	bArm1VertStn4AglDown_00 AT %MX25416.0 : BOOL;
	bArm1VertStn4AglDown_01 AT %MX25416.1 : BOOL;
	bArm1VertStn4AglDown_02 AT %MX25416.2 : BOOL;
	bArm1VertStn4AglDown_03 AT %MX25416.3 : BOOL;
	bArm1VertStn4AglDown_04 AT %MX25416.4 : BOOL;
	bArm1VertStn4AglDown_05 AT %MX25416.5 : BOOL;
	bArm1VertStn4AglDown_06 AT %MX25416.6 : BOOL;
	bArm1VertStn4AglDown_07 AT %MX25416.7 : BOOL;
	bArm1VertStn4AglDown_08 AT %MX25416.8 : BOOL;
	bArm1VertStn4AglDown_09 AT %MX25416.9 : BOOL;
	bArm1VertStn4AglDown_10 AT %MX25416.10 : BOOL;
	bArm1VertStn4AglDown_11 AT %MX25416.11 : BOOL;
	bArm1VertStn4AglDown_12 AT %MX25416.12 : BOOL;
	bArm1VertStn4AglDown_13 AT %MX25416.13 : BOOL;
	bArm1VertStn4AglDown_14 AT %MX25416.14 : BOOL;
	bArm1VertStn4AglDown_15 AT %MX25416.15 : BOOL;
	bArm1VertStn4AglDown_16 AT %MX25416.16 : BOOL;
	bArm1VertStn4AglDown_17 AT %MX25416.17 : BOOL;
	bArm1VertStn4AglDown_18 AT %MX25416.18 : BOOL;
	bArm1VertStn4AglDown_19 AT %MX25416.19 : BOOL;
	bArm1VertStn4AglDown_20 AT %MX25416.20 : BOOL;
	bArm1VertStn4AglDown_21 AT %MX25416.21 : BOOL;
	bArm1VertStn4AglDown_22 AT %MX25416.22 : BOOL;
	bArm1VertStn4AglDown_23 AT %MX25416.23 : BOOL;
	bArm1VertStn4AglDown_24 AT %MX25416.24 : BOOL;
	bArm1VertStn4AglDown_25 AT %MX25416.25 : BOOL;
	bArm1VertStn4AglDown_26 AT %MX25416.26 : BOOL;
	bArm1VertStn4AglDown_27 AT %MX25416.27 : BOOL;
	bArm1VertStn4AglDown_28 AT %MX25416.28 : BOOL;
	bArm1VertStn4AglDown_29 AT %MX25416.29 : BOOL;
	bArm1VertStn4AglDown_30 AT %MX25416.30 : BOOL;
	bArm1VertStn4AglDown_31 AT %MX25416.31 : BOOL;

	bArm1VertStn5AglDown_00 AT %MX25420.0 : BOOL;
	bArm1VertStn5AglDown_01 AT %MX25420.1 : BOOL;
	bArm1VertStn5AglDown_02 AT %MX25420.2 : BOOL;
	bArm1VertStn5AglDown_03 AT %MX25420.3 : BOOL;
	bArm1VertStn5AglDown_04 AT %MX25420.4 : BOOL;
	bArm1VertStn5AglDown_05 AT %MX25420.5 : BOOL;
	bArm1VertStn5AglDown_06 AT %MX25420.6 : BOOL;
	bArm1VertStn5AglDown_07 AT %MX25420.7 : BOOL;
	bArm1VertStn5AglDown_08 AT %MX25420.8 : BOOL;
	bArm1VertStn5AglDown_09 AT %MX25420.9 : BOOL;
	bArm1VertStn5AglDown_10 AT %MX25420.10 : BOOL;
	bArm1VertStn5AglDown_11 AT %MX25420.11 : BOOL;
	bArm1VertStn5AglDown_12 AT %MX25420.12 : BOOL;
	bArm1VertStn5AglDown_13 AT %MX25420.13 : BOOL;
	bArm1VertStn5AglDown_14 AT %MX25420.14 : BOOL;
	bArm1VertStn5AglDown_15 AT %MX25420.15 : BOOL;
	bArm1VertStn5AglDown_16 AT %MX25420.16 : BOOL;
	bArm1VertStn5AglDown_17 AT %MX25420.17 : BOOL;
	bArm1VertStn5AglDown_18 AT %MX25420.18 : BOOL;
	bArm1VertStn5AglDown_19 AT %MX25420.19 : BOOL;
	bArm1VertStn5AglDown_20 AT %MX25420.20 : BOOL;
	bArm1VertStn5AglDown_21 AT %MX25420.21 : BOOL;
	bArm1VertStn5AglDown_22 AT %MX25420.22 : BOOL;
	bArm1VertStn5AglDown_23 AT %MX25420.23 : BOOL;
	bArm1VertStn5AglDown_24 AT %MX25420.24 : BOOL;
	bArm1VertStn5AglDown_25 AT %MX25420.25 : BOOL;
	bArm1VertStn5AglDown_26 AT %MX25420.26 : BOOL;
	bArm1VertStn5AglDown_27 AT %MX25420.27 : BOOL;
	bArm1VertStn5AglDown_28 AT %MX25420.28 : BOOL;
	bArm1VertStn5AglDown_29 AT %MX25420.29 : BOOL;
	bArm1VertStn5AglDown_30 AT %MX25420.30 : BOOL;
	bArm1VertStn5AglDown_31 AT %MX25420.31 : BOOL;

	bArm1VertStn6AglDown_00 AT %MX25424.0 : BOOL;
	bArm1VertStn6AglDown_01 AT %MX25424.1 : BOOL;
	bArm1VertStn6AglDown_02 AT %MX25424.2 : BOOL;
	bArm1VertStn6AglDown_03 AT %MX25424.3 : BOOL;
	bArm1VertStn6AglDown_04 AT %MX25424.4 : BOOL;
	bArm1VertStn6AglDown_05 AT %MX25424.5 : BOOL;
	bArm1VertStn6AglDown_06 AT %MX25424.6 : BOOL;
	bArm1VertStn6AglDown_07 AT %MX25424.7 : BOOL;
	bArm1VertStn6AglDown_08 AT %MX25424.8 : BOOL;
	bArm1VertStn6AglDown_09 AT %MX25424.9 : BOOL;
	bArm1VertStn6AglDown_10 AT %MX25424.10 : BOOL;
	bArm1VertStn6AglDown_11 AT %MX25424.11 : BOOL;
	bArm1VertStn6AglDown_12 AT %MX25424.12 : BOOL;
	bArm1VertStn6AglDown_13 AT %MX25424.13 : BOOL;
	bArm1VertStn6AglDown_14 AT %MX25424.14 : BOOL;
	bArm1VertStn6AglDown_15 AT %MX25424.15 : BOOL;
	bArm1VertStn6AglDown_16 AT %MX25424.16 : BOOL;
	bArm1VertStn6AglDown_17 AT %MX25424.17 : BOOL;
	bArm1VertStn6AglDown_18 AT %MX25424.18 : BOOL;
	bArm1VertStn6AglDown_19 AT %MX25424.19 : BOOL;
	bArm1VertStn6AglDown_20 AT %MX25424.20 : BOOL;
	bArm1VertStn6AglDown_21 AT %MX25424.21 : BOOL;
	bArm1VertStn6AglDown_22 AT %MX25424.22 : BOOL;
	bArm1VertStn6AglDown_23 AT %MX25424.23 : BOOL;
	bArm1VertStn6AglDown_24 AT %MX25424.24 : BOOL;
	bArm1VertStn6AglDown_25 AT %MX25424.25 : BOOL;
	bArm1VertStn6AglDown_26 AT %MX25424.26 : BOOL;
	bArm1VertStn6AglDown_27 AT %MX25424.27 : BOOL;
	bArm1VertStn6AglDown_28 AT %MX25424.28 : BOOL;
	bArm1VertStn6AglDown_29 AT %MX25424.29 : BOOL;
	bArm1VertStn6AglDown_30 AT %MX25424.30 : BOOL;
	bArm1VertStn6AglDown_31 AT %MX25424.31 : BOOL;

	bArm1VertStn7AglDown_00 AT %MX25428.0 : BOOL;
	bArm1VertStn7AglDown_01 AT %MX25428.1 : BOOL;
	bArm1VertStn7AglDown_02 AT %MX25428.2 : BOOL;
	bArm1VertStn7AglDown_03 AT %MX25428.3 : BOOL;
	bArm1VertStn7AglDown_04 AT %MX25428.4 : BOOL;
	bArm1VertStn7AglDown_05 AT %MX25428.5 : BOOL;
	bArm1VertStn7AglDown_06 AT %MX25428.6 : BOOL;
	bArm1VertStn7AglDown_07 AT %MX25428.7 : BOOL;
	bArm1VertStn7AglDown_08 AT %MX25428.8 : BOOL;
	bArm1VertStn7AglDown_09 AT %MX25428.9 : BOOL;
	bArm1VertStn7AglDown_10 AT %MX25428.10 : BOOL;
	bArm1VertStn7AglDown_11 AT %MX25428.11 : BOOL;
	bArm1VertStn7AglDown_12 AT %MX25428.12 : BOOL;
	bArm1VertStn7AglDown_13 AT %MX25428.13 : BOOL;
	bArm1VertStn7AglDown_14 AT %MX25428.14 : BOOL;
	bArm1VertStn7AglDown_15 AT %MX25428.15 : BOOL;
	bArm1VertStn7AglDown_16 AT %MX25428.16 : BOOL;
	bArm1VertStn7AglDown_17 AT %MX25428.17 : BOOL;
	bArm1VertStn7AglDown_18 AT %MX25428.18 : BOOL;
	bArm1VertStn7AglDown_19 AT %MX25428.19 : BOOL;
	bArm1VertStn7AglDown_20 AT %MX25428.20 : BOOL;
	bArm1VertStn7AglDown_21 AT %MX25428.21 : BOOL;
	bArm1VertStn7AglDown_22 AT %MX25428.22 : BOOL;
	bArm1VertStn7AglDown_23 AT %MX25428.23 : BOOL;
	bArm1VertStn7AglDown_24 AT %MX25428.24 : BOOL;
	bArm1VertStn7AglDown_25 AT %MX25428.25 : BOOL;
	bArm1VertStn7AglDown_26 AT %MX25428.26 : BOOL;
	bArm1VertStn7AglDown_27 AT %MX25428.27 : BOOL;
	bArm1VertStn7AglDown_28 AT %MX25428.28 : BOOL;
	bArm1VertStn7AglDown_29 AT %MX25428.29 : BOOL;
	bArm1VertStn7AglDown_30 AT %MX25428.30 : BOOL;
	bArm1VertStn7AglDown_31 AT %MX25428.31 : BOOL;

	bArm1VertStn8AglDown_00 AT %MX25432.0 : BOOL;
	bArm1VertStn8AglDown_01 AT %MX25432.1 : BOOL;
	bArm1VertStn8AglDown_02 AT %MX25432.2 : BOOL;
	bArm1VertStn8AglDown_03 AT %MX25432.3 : BOOL;
	bArm1VertStn8AglDown_04 AT %MX25432.4 : BOOL;
	bArm1VertStn8AglDown_05 AT %MX25432.5 : BOOL;
	bArm1VertStn8AglDown_06 AT %MX25432.6 : BOOL;
	bArm1VertStn8AglDown_07 AT %MX25432.7 : BOOL;
	bArm1VertStn8AglDown_08 AT %MX25432.8 : BOOL;
	bArm1VertStn8AglDown_09 AT %MX25432.9 : BOOL;
	bArm1VertStn8AglDown_10 AT %MX25432.10 : BOOL;
	bArm1VertStn8AglDown_11 AT %MX25432.11 : BOOL;
	bArm1VertStn8AglDown_12 AT %MX25432.12 : BOOL;
	bArm1VertStn8AglDown_13 AT %MX25432.13 : BOOL;
	bArm1VertStn8AglDown_14 AT %MX25432.14 : BOOL;
	bArm1VertStn8AglDown_15 AT %MX25432.15 : BOOL;
	bArm1VertStn8AglDown_16 AT %MX25432.16 : BOOL;
	bArm1VertStn8AglDown_17 AT %MX25432.17 : BOOL;
	bArm1VertStn8AglDown_18 AT %MX25432.18 : BOOL;
	bArm1VertStn8AglDown_19 AT %MX25432.19 : BOOL;
	bArm1VertStn8AglDown_20 AT %MX25432.20 : BOOL;
	bArm1VertStn8AglDown_21 AT %MX25432.21 : BOOL;
	bArm1VertStn8AglDown_22 AT %MX25432.22 : BOOL;
	bArm1VertStn8AglDown_23 AT %MX25432.23 : BOOL;
	bArm1VertStn8AglDown_24 AT %MX25432.24 : BOOL;
	bArm1VertStn8AglDown_25 AT %MX25432.25 : BOOL;
	bArm1VertStn8AglDown_26 AT %MX25432.26 : BOOL;
	bArm1VertStn8AglDown_27 AT %MX25432.27 : BOOL;
	bArm1VertStn8AglDown_28 AT %MX25432.28 : BOOL;
	bArm1VertStn8AglDown_29 AT %MX25432.29 : BOOL;
	bArm1VertStn8AglDown_30 AT %MX25432.30 : BOOL;
	bArm1VertStn8AglDown_31 AT %MX25432.31 : BOOL;

	bArm1VertStn9AglDown_00 AT %MX25436.0 : BOOL;
	bArm1VertStn9AglDown_01 AT %MX25436.1 : BOOL;
	bArm1VertStn9AglDown_02 AT %MX25436.2 : BOOL;
	bArm1VertStn9AglDown_03 AT %MX25436.3 : BOOL;
	bArm1VertStn9AglDown_04 AT %MX25436.4 : BOOL;
	bArm1VertStn9AglDown_05 AT %MX25436.5 : BOOL;
	bArm1VertStn9AglDown_06 AT %MX25436.6 : BOOL;
	bArm1VertStn9AglDown_07 AT %MX25436.7 : BOOL;
	bArm1VertStn9AglDown_08 AT %MX25436.8 : BOOL;
	bArm1VertStn9AglDown_09 AT %MX25436.9 : BOOL;
	bArm1VertStn9AglDown_10 AT %MX25436.10 : BOOL;
	bArm1VertStn9AglDown_11 AT %MX25436.11 : BOOL;
	bArm1VertStn9AglDown_12 AT %MX25436.12 : BOOL;
	bArm1VertStn9AglDown_13 AT %MX25436.13 : BOOL;
	bArm1VertStn9AglDown_14 AT %MX25436.14 : BOOL;
	bArm1VertStn9AglDown_15 AT %MX25436.15 : BOOL;
	bArm1VertStn9AglDown_16 AT %MX25436.16 : BOOL;
	bArm1VertStn9AglDown_17 AT %MX25436.17 : BOOL;
	bArm1VertStn9AglDown_18 AT %MX25436.18 : BOOL;
	bArm1VertStn9AglDown_19 AT %MX25436.19 : BOOL;
	bArm1VertStn9AglDown_20 AT %MX25436.20 : BOOL;
	bArm1VertStn9AglDown_21 AT %MX25436.21 : BOOL;
	bArm1VertStn9AglDown_22 AT %MX25436.22 : BOOL;
	bArm1VertStn9AglDown_23 AT %MX25436.23 : BOOL;
	bArm1VertStn9AglDown_24 AT %MX25436.24 : BOOL;
	bArm1VertStn9AglDown_25 AT %MX25436.25 : BOOL;
	bArm1VertStn9AglDown_26 AT %MX25436.26 : BOOL;
	bArm1VertStn9AglDown_27 AT %MX25436.27 : BOOL;
	bArm1VertStn9AglDown_28 AT %MX25436.28 : BOOL;
	bArm1VertStn9AglDown_29 AT %MX25436.29 : BOOL;
	bArm1VertStn9AglDown_30 AT %MX25436.30 : BOOL;
	bArm1VertStn9AglDown_31 AT %MX25436.31 : BOOL;

	bArm1VertStn10AglDown_00 AT %MX25440.0 : BOOL;
	bArm1VertStn10AglDown_01 AT %MX25440.1 : BOOL;
	bArm1VertStn10AglDown_02 AT %MX25440.2 : BOOL;
	bArm1VertStn10AglDown_03 AT %MX25440.3 : BOOL;
	bArm1VertStn10AglDown_04 AT %MX25440.4 : BOOL;
	bArm1VertStn10AglDown_05 AT %MX25440.5 : BOOL;
	bArm1VertStn10AglDown_06 AT %MX25440.6 : BOOL;
	bArm1VertStn10AglDown_07 AT %MX25440.7 : BOOL;
	bArm1VertStn10AglDown_08 AT %MX25440.8 : BOOL;
	bArm1VertStn10AglDown_09 AT %MX25440.9 : BOOL;
	bArm1VertStn10AglDown_10 AT %MX25440.10 : BOOL;
	bArm1VertStn10AglDown_11 AT %MX25440.11 : BOOL;
	bArm1VertStn10AglDown_12 AT %MX25440.12 : BOOL;
	bArm1VertStn10AglDown_13 AT %MX25440.13 : BOOL;
	bArm1VertStn10AglDown_14 AT %MX25440.14 : BOOL;
	bArm1VertStn10AglDown_15 AT %MX25440.15 : BOOL;
	bArm1VertStn10AglDown_16 AT %MX25440.16 : BOOL;
	bArm1VertStn10AglDown_17 AT %MX25440.17 : BOOL;
	bArm1VertStn10AglDown_18 AT %MX25440.18 : BOOL;
	bArm1VertStn10AglDown_19 AT %MX25440.19 : BOOL;
	bArm1VertStn10AglDown_20 AT %MX25440.20 : BOOL;
	bArm1VertStn10AglDown_21 AT %MX25440.21 : BOOL;
	bArm1VertStn10AglDown_22 AT %MX25440.22 : BOOL;
	bArm1VertStn10AglDown_23 AT %MX25440.23 : BOOL;
	bArm1VertStn10AglDown_24 AT %MX25440.24 : BOOL;
	bArm1VertStn10AglDown_25 AT %MX25440.25 : BOOL;
	bArm1VertStn10AglDown_26 AT %MX25440.26 : BOOL;
	bArm1VertStn10AglDown_27 AT %MX25440.27 : BOOL;
	bArm1VertStn10AglDown_28 AT %MX25440.28 : BOOL;
	bArm1VertStn10AglDown_29 AT %MX25440.29 : BOOL;
	bArm1VertStn10AglDown_30 AT %MX25440.30 : BOOL;
	bArm1VertStn10AglDown_31 AT %MX25440.31 : BOOL;

	bArm1VertStn11AglDown_00 AT %MX25444.0 : BOOL;
	bArm1VertStn11AglDown_01 AT %MX25444.1 : BOOL;
	bArm1VertStn11AglDown_02 AT %MX25444.2 : BOOL;
	bArm1VertStn11AglDown_03 AT %MX25444.3 : BOOL;
	bArm1VertStn11AglDown_04 AT %MX25444.4 : BOOL;
	bArm1VertStn11AglDown_05 AT %MX25444.5 : BOOL;
	bArm1VertStn11AglDown_06 AT %MX25444.6 : BOOL;
	bArm1VertStn11AglDown_07 AT %MX25444.7 : BOOL;
	bArm1VertStn11AglDown_08 AT %MX25444.8 : BOOL;
	bArm1VertStn11AglDown_09 AT %MX25444.9 : BOOL;
	bArm1VertStn11AglDown_10 AT %MX25444.10 : BOOL;
	bArm1VertStn11AglDown_11 AT %MX25444.11 : BOOL;
	bArm1VertStn11AglDown_12 AT %MX25444.12 : BOOL;
	bArm1VertStn11AglDown_13 AT %MX25444.13 : BOOL;
	bArm1VertStn11AglDown_14 AT %MX25444.14 : BOOL;
	bArm1VertStn11AglDown_15 AT %MX25444.15 : BOOL;
	bArm1VertStn11AglDown_16 AT %MX25444.16 : BOOL;
	bArm1VertStn11AglDown_17 AT %MX25444.17 : BOOL;
	bArm1VertStn11AglDown_18 AT %MX25444.18 : BOOL;
	bArm1VertStn11AglDown_19 AT %MX25444.19 : BOOL;
	bArm1VertStn11AglDown_20 AT %MX25444.20 : BOOL;
	bArm1VertStn11AglDown_21 AT %MX25444.21 : BOOL;
	bArm1VertStn11AglDown_22 AT %MX25444.22 : BOOL;
	bArm1VertStn11AglDown_23 AT %MX25444.23 : BOOL;
	bArm1VertStn11AglDown_24 AT %MX25444.24 : BOOL;
	bArm1VertStn11AglDown_25 AT %MX25444.25 : BOOL;
	bArm1VertStn11AglDown_26 AT %MX25444.26 : BOOL;
	bArm1VertStn11AglDown_27 AT %MX25444.27 : BOOL;
	bArm1VertStn11AglDown_28 AT %MX25444.28 : BOOL;
	bArm1VertStn11AglDown_29 AT %MX25444.29 : BOOL;
	bArm1VertStn11AglDown_30 AT %MX25444.30 : BOOL;
	bArm1VertStn11AglDown_31 AT %MX25444.31 : BOOL;

	bArm1VertStn12AglDown_00 AT %MX25448.0 : BOOL;
	bArm1VertStn12AglDown_01 AT %MX25448.1 : BOOL;
	bArm1VertStn12AglDown_02 AT %MX25448.2 : BOOL;
	bArm1VertStn12AglDown_03 AT %MX25448.3 : BOOL;
	bArm1VertStn12AglDown_04 AT %MX25448.4 : BOOL;
	bArm1VertStn12AglDown_05 AT %MX25448.5 : BOOL;
	bArm1VertStn12AglDown_06 AT %MX25448.6 : BOOL;
	bArm1VertStn12AglDown_07 AT %MX25448.7 : BOOL;
	bArm1VertStn12AglDown_08 AT %MX25448.8 : BOOL;
	bArm1VertStn12AglDown_09 AT %MX25448.9 : BOOL;
	bArm1VertStn12AglDown_10 AT %MX25448.10 : BOOL;
	bArm1VertStn12AglDown_11 AT %MX25448.11 : BOOL;
	bArm1VertStn12AglDown_12 AT %MX25448.12 : BOOL;
	bArm1VertStn12AglDown_13 AT %MX25448.13 : BOOL;
	bArm1VertStn12AglDown_14 AT %MX25448.14 : BOOL;
	bArm1VertStn12AglDown_15 AT %MX25448.15 : BOOL;
	bArm1VertStn12AglDown_16 AT %MX25448.16 : BOOL;
	bArm1VertStn12AglDown_17 AT %MX25448.17 : BOOL;
	bArm1VertStn12AglDown_18 AT %MX25448.18 : BOOL;
	bArm1VertStn12AglDown_19 AT %MX25448.19 : BOOL;
	bArm1VertStn12AglDown_20 AT %MX25448.20 : BOOL;
	bArm1VertStn12AglDown_21 AT %MX25448.21 : BOOL;
	bArm1VertStn12AglDown_22 AT %MX25448.22 : BOOL;
	bArm1VertStn12AglDown_23 AT %MX25448.23 : BOOL;
	bArm1VertStn12AglDown_24 AT %MX25448.24 : BOOL;
	bArm1VertStn12AglDown_25 AT %MX25448.25 : BOOL;
	bArm1VertStn12AglDown_26 AT %MX25448.26 : BOOL;
	bArm1VertStn12AglDown_27 AT %MX25448.27 : BOOL;
	bArm1VertStn12AglDown_28 AT %MX25448.28 : BOOL;
	bArm1VertStn12AglDown_29 AT %MX25448.29 : BOOL;
	bArm1VertStn12AglDown_30 AT %MX25448.30 : BOOL;
	bArm1VertStn12AglDown_31 AT %MX25448.31 : BOOL;


(* xxxxxxxxxxxxxxxxxxxxxxxxxxxxxxxxxxxxxxx Vert xxxxxxxxxxxxxxxxxxxxxxxxxxxxxxxxxxxxxxx*)
(*========= Down BOOL LINK with %MX25500-MX25599 =========*)

	bArm1VertLD1Down_00 AT %MX25552.0 : BOOL;
	bArm1VertLD1Down_01 AT %MX25552.1 : BOOL;
	bArm1VertLD1Down_02 AT %MX25552.2 : BOOL;
	bArm1VertLD1Down_03 AT %MX25552.3 : BOOL;
	bArm1VertLD1Down_04 AT %MX25552.4 : BOOL;
	bArm1VertLD1Down_05 AT %MX25552.5 : BOOL;
	bArm1VertLD1Down_06 AT %MX25552.6 : BOOL;
	bArm1VertLD1Down_07 AT %MX25552.7 : BOOL;
	bArm1VertLD1Down_08 AT %MX25552.8 : BOOL;
	bArm1VertLD1Down_09 AT %MX25552.9 : BOOL;
	bArm1VertLD1Down_10 AT %MX25552.10 : BOOL;
	bArm1VertLD1Down_11 AT %MX25552.11 : BOOL;
	bArm1VertLD1Down_12 AT %MX25552.12 : BOOL;
	bArm1VertLD1Down_13 AT %MX25552.13 : BOOL;
	bArm1VertLD1Down_14 AT %MX25552.14 : BOOL;
	bArm1VertLD1Down_15 AT %MX25552.15 : BOOL;
	bArm1VertLD1Down_16 AT %MX25552.16 : BOOL;
	bArm1VertLD1Down_17 AT %MX25552.17 : BOOL;
	bArm1VertLD1Down_18 AT %MX25552.18 : BOOL;
	bArm1VertLD1Down_19 AT %MX25552.19 : BOOL;
	bArm1VertLD1Down_20 AT %MX25552.20 : BOOL;
	bArm1VertLD1Down_21 AT %MX25552.21 : BOOL;
	bArm1VertLD1Down_22 AT %MX25552.22 : BOOL;
	bArm1VertLD1Down_23 AT %MX25552.23 : BOOL;
	bArm1VertLD1Down_24 AT %MX25552.24 : BOOL;
	bArm1VertLD1Down_25 AT %MX25552.25 : BOOL;
	bArm1VertLD1Down_26 AT %MX25552.26 : BOOL;
	bArm1VertLD1Down_27 AT %MX25552.27 : BOOL;
	bArm1VertLD1Down_28 AT %MX25552.28 : BOOL;
	bArm1VertLD1Down_29 AT %MX25552.29 : BOOL;
	bArm1VertLD1Down_30 AT %MX25552.30 : BOOL;
	bArm1VertLD1Down_31 AT %MX25552.31 : BOOL;

	bArm1VertULD1Down_00 AT %MX25556.0 : BOOL;
	bArm1VertULD1Down_01 AT %MX25556.1 : BOOL;
	bArm1VertULD1Down_02 AT %MX25556.2 : BOOL;
	bArm1VertULD1Down_03 AT %MX25556.3 : BOOL;
	bArm1VertULD1Down_04 AT %MX25556.4 : BOOL;
	bArm1VertULD1Down_05 AT %MX25556.5 : BOOL;
	bArm1VertULD1Down_06 AT %MX25556.6 : BOOL;
	bArm1VertULD1Down_07 AT %MX25556.7 : BOOL;
	bArm1VertULD1Down_08 AT %MX25556.8 : BOOL;
	bArm1VertULD1Down_09 AT %MX25556.9 : BOOL;
	bArm1VertULD1Down_10 AT %MX25556.10 : BOOL;
	bArm1VertULD1Down_11 AT %MX25556.11 : BOOL;
	bArm1VertULD1Down_12 AT %MX25556.12 : BOOL;
	bArm1VertULD1Down_13 AT %MX25556.13 : BOOL;
	bArm1VertULD1Down_14 AT %MX25556.14 : BOOL;
	bArm1VertULD1Down_15 AT %MX25556.15 : BOOL;
	bArm1VertULD1Down_16 AT %MX25556.16 : BOOL;
	bArm1VertULD1Down_17 AT %MX25556.17 : BOOL;
	bArm1VertULD1Down_18 AT %MX25556.18 : BOOL;
	bArm1VertULD1Down_19 AT %MX25556.19 : BOOL;
	bArm1VertULD1Down_20 AT %MX25556.20 : BOOL;
	bArm1VertULD1Down_21 AT %MX25556.21 : BOOL;
	bArm1VertULD1Down_22 AT %MX25556.22 : BOOL;
	bArm1VertULD1Down_23 AT %MX25556.23 : BOOL;
	bArm1VertULD1Down_24 AT %MX25556.24 : BOOL;
	bArm1VertULD1Down_25 AT %MX25556.25 : BOOL;
	bArm1VertULD1Down_26 AT %MX25556.26 : BOOL;
	bArm1VertULD1Down_27 AT %MX25556.27 : BOOL;
	bArm1VertULD1Down_28 AT %MX25556.28 : BOOL;
	bArm1VertULD1Down_29 AT %MX25556.29 : BOOL;
	bArm1VertULD1Down_30 AT %MX25556.30 : BOOL;
	bArm1VertULD1Down_31 AT %MX25556.31 : BOOL;

	bArm1VertStn1Down_00 AT %MX25504.0 : BOOL;
	bArm1VertStn1Down_01 AT %MX25504.1 : BOOL;
	bArm1VertStn1Down_02 AT %MX25504.2 : BOOL;
	bArm1VertStn1Down_03 AT %MX25504.3 : BOOL;
	bArm1VertStn1Down_04 AT %MX25504.4 : BOOL;
	bArm1VertStn1Down_05 AT %MX25504.5 : BOOL;
	bArm1VertStn1Down_06 AT %MX25504.6 : BOOL;
	bArm1VertStn1Down_07 AT %MX25504.7 : BOOL;
	bArm1VertStn1Down_08 AT %MX25504.8 : BOOL;
	bArm1VertStn1Down_09 AT %MX25504.9 : BOOL;
	bArm1VertStn1Down_10 AT %MX25504.10 : BOOL;
	bArm1VertStn1Down_11 AT %MX25504.11 : BOOL;
	bArm1VertStn1Down_12 AT %MX25504.12 : BOOL;
	bArm1VertStn1Down_13 AT %MX25504.13 : BOOL;
	bArm1VertStn1Down_14 AT %MX25504.14 : BOOL;
	bArm1VertStn1Down_15 AT %MX25504.15 : BOOL;
	bArm1VertStn1Down_16 AT %MX25504.16 : BOOL;
	bArm1VertStn1Down_17 AT %MX25504.17 : BOOL;
	bArm1VertStn1Down_18 AT %MX25504.18 : BOOL;
	bArm1VertStn1Down_19 AT %MX25504.19 : BOOL;
	bArm1VertStn1Down_20 AT %MX25504.20 : BOOL;
	bArm1VertStn1Down_21 AT %MX25504.21 : BOOL;
	bArm1VertStn1Down_22 AT %MX25504.22 : BOOL;
	bArm1VertStn1Down_23 AT %MX25504.23 : BOOL;
	bArm1VertStn1Down_24 AT %MX25504.24 : BOOL;
	bArm1VertStn1Down_25 AT %MX25504.25 : BOOL;
	bArm1VertStn1Down_26 AT %MX25504.26 : BOOL;
	bArm1VertStn1Down_27 AT %MX25504.27 : BOOL;
	bArm1VertStn1Down_28 AT %MX25504.28 : BOOL;
	bArm1VertStn1Down_29 AT %MX25504.29 : BOOL;
	bArm1VertStn1Down_30 AT %MX25504.30 : BOOL;
	bArm1VertStn1Down_31 AT %MX25504.31 : BOOL;

	bArm1VertStn2Down_00 AT %MX25508.0 : BOOL;
	bArm1VertStn2Down_01 AT %MX25508.1 : BOOL;
	bArm1VertStn2Down_02 AT %MX25508.2 : BOOL;
	bArm1VertStn2Down_03 AT %MX25508.3 : BOOL;
	bArm1VertStn2Down_04 AT %MX25508.4 : BOOL;
	bArm1VertStn2Down_05 AT %MX25508.5 : BOOL;
	bArm1VertStn2Down_06 AT %MX25508.6 : BOOL;
	bArm1VertStn2Down_07 AT %MX25508.7 : BOOL;
	bArm1VertStn2Down_08 AT %MX25508.8 : BOOL;
	bArm1VertStn2Down_09 AT %MX25508.9 : BOOL;
	bArm1VertStn2Down_10 AT %MX25508.10 : BOOL;
	bArm1VertStn2Down_11 AT %MX25508.11 : BOOL;
	bArm1VertStn2Down_12 AT %MX25508.12 : BOOL;
	bArm1VertStn2Down_13 AT %MX25508.13 : BOOL;
	bArm1VertStn2Down_14 AT %MX25508.14 : BOOL;
	bArm1VertStn2Down_15 AT %MX25508.15 : BOOL;
	bArm1VertStn2Down_16 AT %MX25508.16 : BOOL;
	bArm1VertStn2Down_17 AT %MX25508.17 : BOOL;
	bArm1VertStn2Down_18 AT %MX25508.18 : BOOL;
	bArm1VertStn2Down_19 AT %MX25508.19 : BOOL;
	bArm1VertStn2Down_20 AT %MX25508.20 : BOOL;
	bArm1VertStn2Down_21 AT %MX25508.21 : BOOL;
	bArm1VertStn2Down_22 AT %MX25508.22 : BOOL;
	bArm1VertStn2Down_23 AT %MX25508.23 : BOOL;
	bArm1VertStn2Down_24 AT %MX25508.24 : BOOL;
	bArm1VertStn2Down_25 AT %MX25508.25 : BOOL;
	bArm1VertStn2Down_26 AT %MX25508.26 : BOOL;
	bArm1VertStn2Down_27 AT %MX25508.27 : BOOL;
	bArm1VertStn2Down_28 AT %MX25508.28 : BOOL;
	bArm1VertStn2Down_29 AT %MX25508.29 : BOOL;
	bArm1VertStn2Down_30 AT %MX25508.30 : BOOL;
	bArm1VertStn2Down_31 AT %MX25508.31 : BOOL;

	bArm1VertStn3Down_00 AT %MX25512.0 : BOOL;
	bArm1VertStn3Down_01 AT %MX25512.1 : BOOL;
	bArm1VertStn3Down_02 AT %MX25512.2 : BOOL;
	bArm1VertStn3Down_03 AT %MX25512.3 : BOOL;
	bArm1VertStn3Down_04 AT %MX25512.4 : BOOL;
	bArm1VertStn3Down_05 AT %MX25512.5 : BOOL;
	bArm1VertStn3Down_06 AT %MX25512.6 : BOOL;
	bArm1VertStn3Down_07 AT %MX25512.7 : BOOL;
	bArm1VertStn3Down_08 AT %MX25512.8 : BOOL;
	bArm1VertStn3Down_09 AT %MX25512.9 : BOOL;
	bArm1VertStn3Down_10 AT %MX25512.10 : BOOL;
	bArm1VertStn3Down_11 AT %MX25512.11 : BOOL;
	bArm1VertStn3Down_12 AT %MX25512.12 : BOOL;
	bArm1VertStn3Down_13 AT %MX25512.13 : BOOL;
	bArm1VertStn3Down_14 AT %MX25512.14 : BOOL;
	bArm1VertStn3Down_15 AT %MX25512.15 : BOOL;
	bArm1VertStn3Down_16 AT %MX25512.16 : BOOL;
	bArm1VertStn3Down_17 AT %MX25512.17 : BOOL;
	bArm1VertStn3Down_18 AT %MX25512.18 : BOOL;
	bArm1VertStn3Down_19 AT %MX25512.19 : BOOL;
	bArm1VertStn3Down_20 AT %MX25512.20 : BOOL;
	bArm1VertStn3Down_21 AT %MX25512.21 : BOOL;
	bArm1VertStn3Down_22 AT %MX25512.22 : BOOL;
	bArm1VertStn3Down_23 AT %MX25512.23 : BOOL;
	bArm1VertStn3Down_24 AT %MX25512.24 : BOOL;
	bArm1VertStn3Down_25 AT %MX25512.25 : BOOL;
	bArm1VertStn3Down_26 AT %MX25512.26 : BOOL;
	bArm1VertStn3Down_27 AT %MX25512.27 : BOOL;
	bArm1VertStn3Down_28 AT %MX25512.28 : BOOL;
	bArm1VertStn3Down_29 AT %MX25512.29 : BOOL;
	bArm1VertStn3Down_30 AT %MX25512.30 : BOOL;
	bArm1VertStn3Down_31 AT %MX25512.31 : BOOL;

	bArm1VertStn4Down_00 AT %MX25516.0 : BOOL;
	bArm1VertStn4Down_01 AT %MX25516.1 : BOOL;
	bArm1VertStn4Down_02 AT %MX25516.2 : BOOL;
	bArm1VertStn4Down_03 AT %MX25516.3 : BOOL;
	bArm1VertStn4Down_04 AT %MX25516.4 : BOOL;
	bArm1VertStn4Down_05 AT %MX25516.5 : BOOL;
	bArm1VertStn4Down_06 AT %MX25516.6 : BOOL;
	bArm1VertStn4Down_07 AT %MX25516.7 : BOOL;
	bArm1VertStn4Down_08 AT %MX25516.8 : BOOL;
	bArm1VertStn4Down_09 AT %MX25516.9 : BOOL;
	bArm1VertStn4Down_10 AT %MX25516.10 : BOOL;
	bArm1VertStn4Down_11 AT %MX25516.11 : BOOL;
	bArm1VertStn4Down_12 AT %MX25516.12 : BOOL;
	bArm1VertStn4Down_13 AT %MX25516.13 : BOOL;
	bArm1VertStn4Down_14 AT %MX25516.14 : BOOL;
	bArm1VertStn4Down_15 AT %MX25516.15 : BOOL;
	bArm1VertStn4Down_16 AT %MX25516.16 : BOOL;
	bArm1VertStn4Down_17 AT %MX25516.17 : BOOL;
	bArm1VertStn4Down_18 AT %MX25516.18 : BOOL;
	bArm1VertStn4Down_19 AT %MX25516.19 : BOOL;
	bArm1VertStn4Down_20 AT %MX25516.20 : BOOL;
	bArm1VertStn4Down_21 AT %MX25516.21 : BOOL;
	bArm1VertStn4Down_22 AT %MX25516.22 : BOOL;
	bArm1VertStn4Down_23 AT %MX25516.23 : BOOL;
	bArm1VertStn4Down_24 AT %MX25516.24 : BOOL;
	bArm1VertStn4Down_25 AT %MX25516.25 : BOOL;
	bArm1VertStn4Down_26 AT %MX25516.26 : BOOL;
	bArm1VertStn4Down_27 AT %MX25516.27 : BOOL;
	bArm1VertStn4Down_28 AT %MX25516.28 : BOOL;
	bArm1VertStn4Down_29 AT %MX25516.29 : BOOL;
	bArm1VertStn4Down_30 AT %MX25516.30 : BOOL;
	bArm1VertStn4Down_31 AT %MX25516.31 : BOOL;

	bArm1VertStn5Down_00 AT %MX25520.0 : BOOL;
	bArm1VertStn5Down_01 AT %MX25520.1 : BOOL;
	bArm1VertStn5Down_02 AT %MX25520.2 : BOOL;
	bArm1VertStn5Down_03 AT %MX25520.3 : BOOL;
	bArm1VertStn5Down_04 AT %MX25520.4 : BOOL;
	bArm1VertStn5Down_05 AT %MX25520.5 : BOOL;
	bArm1VertStn5Down_06 AT %MX25520.6 : BOOL;
	bArm1VertStn5Down_07 AT %MX25520.7 : BOOL;
	bArm1VertStn5Down_08 AT %MX25520.8 : BOOL;
	bArm1VertStn5Down_09 AT %MX25520.9 : BOOL;
	bArm1VertStn5Down_10 AT %MX25520.10 : BOOL;
	bArm1VertStn5Down_11 AT %MX25520.11 : BOOL;
	bArm1VertStn5Down_12 AT %MX25520.12 : BOOL;
	bArm1VertStn5Down_13 AT %MX25520.13 : BOOL;
	bArm1VertStn5Down_14 AT %MX25520.14 : BOOL;
	bArm1VertStn5Down_15 AT %MX25520.15 : BOOL;
	bArm1VertStn5Down_16 AT %MX25520.16 : BOOL;
	bArm1VertStn5Down_17 AT %MX25520.17 : BOOL;
	bArm1VertStn5Down_18 AT %MX25520.18 : BOOL;
	bArm1VertStn5Down_19 AT %MX25520.19 : BOOL;
	bArm1VertStn5Down_20 AT %MX25520.20 : BOOL;
	bArm1VertStn5Down_21 AT %MX25520.21 : BOOL;
	bArm1VertStn5Down_22 AT %MX25520.22 : BOOL;
	bArm1VertStn5Down_23 AT %MX25520.23 : BOOL;
	bArm1VertStn5Down_24 AT %MX25520.24 : BOOL;
	bArm1VertStn5Down_25 AT %MX25520.25 : BOOL;
	bArm1VertStn5Down_26 AT %MX25520.26 : BOOL;
	bArm1VertStn5Down_27 AT %MX25520.27 : BOOL;
	bArm1VertStn5Down_28 AT %MX25520.28 : BOOL;
	bArm1VertStn5Down_29 AT %MX25520.29 : BOOL;
	bArm1VertStn5Down_30 AT %MX25520.30 : BOOL;
	bArm1VertStn5Down_31 AT %MX25520.31 : BOOL;

	bArm1VertStn6Down_00 AT %MX25524.0 : BOOL;
	bArm1VertStn6Down_01 AT %MX25524.1 : BOOL;
	bArm1VertStn6Down_02 AT %MX25524.2 : BOOL;
	bArm1VertStn6Down_03 AT %MX25524.3 : BOOL;
	bArm1VertStn6Down_04 AT %MX25524.4 : BOOL;
	bArm1VertStn6Down_05 AT %MX25524.5 : BOOL;
	bArm1VertStn6Down_06 AT %MX25524.6 : BOOL;
	bArm1VertStn6Down_07 AT %MX25524.7 : BOOL;
	bArm1VertStn6Down_08 AT %MX25524.8 : BOOL;
	bArm1VertStn6Down_09 AT %MX25524.9 : BOOL;
	bArm1VertStn6Down_10 AT %MX25524.10 : BOOL;
	bArm1VertStn6Down_11 AT %MX25524.11 : BOOL;
	bArm1VertStn6Down_12 AT %MX25524.12 : BOOL;
	bArm1VertStn6Down_13 AT %MX25524.13 : BOOL;
	bArm1VertStn6Down_14 AT %MX25524.14 : BOOL;
	bArm1VertStn6Down_15 AT %MX25524.15 : BOOL;
	bArm1VertStn6Down_16 AT %MX25524.16 : BOOL;
	bArm1VertStn6Down_17 AT %MX25524.17 : BOOL;
	bArm1VertStn6Down_18 AT %MX25524.18 : BOOL;
	bArm1VertStn6Down_19 AT %MX25524.19 : BOOL;
	bArm1VertStn6Down_20 AT %MX25524.20 : BOOL;
	bArm1VertStn6Down_21 AT %MX25524.21 : BOOL;
	bArm1VertStn6Down_22 AT %MX25524.22 : BOOL;
	bArm1VertStn6Down_23 AT %MX25524.23 : BOOL;
	bArm1VertStn6Down_24 AT %MX25524.24 : BOOL;
	bArm1VertStn6Down_25 AT %MX25524.25 : BOOL;
	bArm1VertStn6Down_26 AT %MX25524.26 : BOOL;
	bArm1VertStn6Down_27 AT %MX25524.27 : BOOL;
	bArm1VertStn6Down_28 AT %MX25524.28 : BOOL;
	bArm1VertStn6Down_29 AT %MX25524.29 : BOOL;
	bArm1VertStn6Down_30 AT %MX25524.30 : BOOL;
	bArm1VertStn6Down_31 AT %MX25524.31 : BOOL;

	bArm1VertStn7Down_00 AT %MX25528.0 : BOOL;
	bArm1VertStn7Down_01 AT %MX25528.1 : BOOL;
	bArm1VertStn7Down_02 AT %MX25528.2 : BOOL;
	bArm1VertStn7Down_03 AT %MX25528.3 : BOOL;
	bArm1VertStn7Down_04 AT %MX25528.4 : BOOL;
	bArm1VertStn7Down_05 AT %MX25528.5 : BOOL;
	bArm1VertStn7Down_06 AT %MX25528.6 : BOOL;
	bArm1VertStn7Down_07 AT %MX25528.7 : BOOL;
	bArm1VertStn7Down_08 AT %MX25528.8 : BOOL;
	bArm1VertStn7Down_09 AT %MX25528.9 : BOOL;
	bArm1VertStn7Down_10 AT %MX25528.10 : BOOL;
	bArm1VertStn7Down_11 AT %MX25528.11 : BOOL;
	bArm1VertStn7Down_12 AT %MX25528.12 : BOOL;
	bArm1VertStn7Down_13 AT %MX25528.13 : BOOL;
	bArm1VertStn7Down_14 AT %MX25528.14 : BOOL;
	bArm1VertStn7Down_15 AT %MX25528.15 : BOOL;
	bArm1VertStn7Down_16 AT %MX25528.16 : BOOL;
	bArm1VertStn7Down_17 AT %MX25528.17 : BOOL;
	bArm1VertStn7Down_18 AT %MX25528.18 : BOOL;
	bArm1VertStn7Down_19 AT %MX25528.19 : BOOL;
	bArm1VertStn7Down_20 AT %MX25528.20 : BOOL;
	bArm1VertStn7Down_21 AT %MX25528.21 : BOOL;
	bArm1VertStn7Down_22 AT %MX25528.22 : BOOL;
	bArm1VertStn7Down_23 AT %MX25528.23 : BOOL;
	bArm1VertStn7Down_24 AT %MX25528.24 : BOOL;
	bArm1VertStn7Down_25 AT %MX25528.25 : BOOL;
	bArm1VertStn7Down_26 AT %MX25528.26 : BOOL;
	bArm1VertStn7Down_27 AT %MX25528.27 : BOOL;
	bArm1VertStn7Down_28 AT %MX25528.28 : BOOL;
	bArm1VertStn7Down_29 AT %MX25528.29 : BOOL;
	bArm1VertStn7Down_30 AT %MX25528.30 : BOOL;
	bArm1VertStn7Down_31 AT %MX25528.31 : BOOL;

	bArm1VertStn8Down_00 AT %MX25532.0 : BOOL;
	bArm1VertStn8Down_01 AT %MX25532.1 : BOOL;
	bArm1VertStn8Down_02 AT %MX25532.2 : BOOL;
	bArm1VertStn8Down_03 AT %MX25532.3 : BOOL;
	bArm1VertStn8Down_04 AT %MX25532.4 : BOOL;
	bArm1VertStn8Down_05 AT %MX25532.5 : BOOL;
	bArm1VertStn8Down_06 AT %MX25532.6 : BOOL;
	bArm1VertStn8Down_07 AT %MX25532.7 : BOOL;
	bArm1VertStn8Down_08 AT %MX25532.8 : BOOL;
	bArm1VertStn8Down_09 AT %MX25532.9 : BOOL;
	bArm1VertStn8Down_10 AT %MX25532.10 : BOOL;
	bArm1VertStn8Down_11 AT %MX25532.11 : BOOL;
	bArm1VertStn8Down_12 AT %MX25532.12 : BOOL;
	bArm1VertStn8Down_13 AT %MX25532.13 : BOOL;
	bArm1VertStn8Down_14 AT %MX25532.14 : BOOL;
	bArm1VertStn8Down_15 AT %MX25532.15 : BOOL;
	bArm1VertStn8Down_16 AT %MX25532.16 : BOOL;
	bArm1VertStn8Down_17 AT %MX25532.17 : BOOL;
	bArm1VertStn8Down_18 AT %MX25532.18 : BOOL;
	bArm1VertStn8Down_19 AT %MX25532.19 : BOOL;
	bArm1VertStn8Down_20 AT %MX25532.20 : BOOL;
	bArm1VertStn8Down_21 AT %MX25532.21 : BOOL;
	bArm1VertStn8Down_22 AT %MX25532.22 : BOOL;
	bArm1VertStn8Down_23 AT %MX25532.23 : BOOL;
	bArm1VertStn8Down_24 AT %MX25532.24 : BOOL;
	bArm1VertStn8Down_25 AT %MX25532.25 : BOOL;
	bArm1VertStn8Down_26 AT %MX25532.26 : BOOL;
	bArm1VertStn8Down_27 AT %MX25532.27 : BOOL;
	bArm1VertStn8Down_28 AT %MX25532.28 : BOOL;
	bArm1VertStn8Down_29 AT %MX25532.29 : BOOL;
	bArm1VertStn8Down_30 AT %MX25532.30 : BOOL;
	bArm1VertStn8Down_31 AT %MX25532.31 : BOOL;

	bArm1VertStn9Down_00 AT %MX25536.0 : BOOL;
	bArm1VertStn9Down_01 AT %MX25536.1 : BOOL;
	bArm1VertStn9Down_02 AT %MX25536.2 : BOOL;
	bArm1VertStn9Down_03 AT %MX25536.3 : BOOL;
	bArm1VertStn9Down_04 AT %MX25536.4 : BOOL;
	bArm1VertStn9Down_05 AT %MX25536.5 : BOOL;
	bArm1VertStn9Down_06 AT %MX25536.6 : BOOL;
	bArm1VertStn9Down_07 AT %MX25536.7 : BOOL;
	bArm1VertStn9Down_08 AT %MX25536.8 : BOOL;
	bArm1VertStn9Down_09 AT %MX25536.9 : BOOL;
	bArm1VertStn9Down_10 AT %MX25536.10 : BOOL;
	bArm1VertStn9Down_11 AT %MX25536.11 : BOOL;
	bArm1VertStn9Down_12 AT %MX25536.12 : BOOL;
	bArm1VertStn9Down_13 AT %MX25536.13 : BOOL;
	bArm1VertStn9Down_14 AT %MX25536.14 : BOOL;
	bArm1VertStn9Down_15 AT %MX25536.15 : BOOL;
	bArm1VertStn9Down_16 AT %MX25536.16 : BOOL;
	bArm1VertStn9Down_17 AT %MX25536.17 : BOOL;
	bArm1VertStn9Down_18 AT %MX25536.18 : BOOL;
	bArm1VertStn9Down_19 AT %MX25536.19 : BOOL;
	bArm1VertStn9Down_20 AT %MX25536.20 : BOOL;
	bArm1VertStn9Down_21 AT %MX25536.21 : BOOL;
	bArm1VertStn9Down_22 AT %MX25536.22 : BOOL;
	bArm1VertStn9Down_23 AT %MX25536.23 : BOOL;
	bArm1VertStn9Down_24 AT %MX25536.24 : BOOL;
	bArm1VertStn9Down_25 AT %MX25536.25 : BOOL;
	bArm1VertStn9Down_26 AT %MX25536.26 : BOOL;
	bArm1VertStn9Down_27 AT %MX25536.27 : BOOL;
	bArm1VertStn9Down_28 AT %MX25536.28 : BOOL;
	bArm1VertStn9Down_29 AT %MX25536.29 : BOOL;
	bArm1VertStn9Down_30 AT %MX25536.30 : BOOL;
	bArm1VertStn9Down_31 AT %MX25536.31 : BOOL;

	bArm1VertStn10Down_00 AT %MX25540.0 : BOOL;
	bArm1VertStn10Down_01 AT %MX25540.1 : BOOL;
	bArm1VertStn10Down_02 AT %MX25540.2 : BOOL;
	bArm1VertStn10Down_03 AT %MX25540.3 : BOOL;
	bArm1VertStn10Down_04 AT %MX25540.4 : BOOL;
	bArm1VertStn10Down_05 AT %MX25540.5 : BOOL;
	bArm1VertStn10Down_06 AT %MX25540.6 : BOOL;
	bArm1VertStn10Down_07 AT %MX25540.7 : BOOL;
	bArm1VertStn10Down_08 AT %MX25540.8 : BOOL;
	bArm1VertStn10Down_09 AT %MX25540.9 : BOOL;
	bArm1VertStn10Down_10 AT %MX25540.10 : BOOL;
	bArm1VertStn10Down_11 AT %MX25540.11 : BOOL;
	bArm1VertStn10Down_12 AT %MX25540.12 : BOOL;
	bArm1VertStn10Down_13 AT %MX25540.13 : BOOL;
	bArm1VertStn10Down_14 AT %MX25540.14 : BOOL;
	bArm1VertStn10Down_15 AT %MX25540.15 : BOOL;
	bArm1VertStn10Down_16 AT %MX25540.16 : BOOL;
	bArm1VertStn10Down_17 AT %MX25540.17 : BOOL;
	bArm1VertStn10Down_18 AT %MX25540.18 : BOOL;
	bArm1VertStn10Down_19 AT %MX25540.19 : BOOL;
	bArm1VertStn10Down_20 AT %MX25540.20 : BOOL;
	bArm1VertStn10Down_21 AT %MX25540.21 : BOOL;
	bArm1VertStn10Down_22 AT %MX25540.22 : BOOL;
	bArm1VertStn10Down_23 AT %MX25540.23 : BOOL;
	bArm1VertStn10Down_24 AT %MX25540.24 : BOOL;
	bArm1VertStn10Down_25 AT %MX25540.25 : BOOL;
	bArm1VertStn10Down_26 AT %MX25540.26 : BOOL;
	bArm1VertStn10Down_27 AT %MX25540.27 : BOOL;
	bArm1VertStn10Down_28 AT %MX25540.28 : BOOL;
	bArm1VertStn10Down_29 AT %MX25540.29 : BOOL;
	bArm1VertStn10Down_30 AT %MX25540.30 : BOOL;
	bArm1VertStn10Down_31 AT %MX25540.31 : BOOL;

	bArm1VertStn11Down_00 AT %MX25544.0 : BOOL;
	bArm1VertStn11Down_01 AT %MX25544.1 : BOOL;
	bArm1VertStn11Down_02 AT %MX25544.2 : BOOL;
	bArm1VertStn11Down_03 AT %MX25544.3 : BOOL;
	bArm1VertStn11Down_04 AT %MX25544.4 : BOOL;
	bArm1VertStn11Down_05 AT %MX25544.5 : BOOL;
	bArm1VertStn11Down_06 AT %MX25544.6 : BOOL;
	bArm1VertStn11Down_07 AT %MX25544.7 : BOOL;
	bArm1VertStn11Down_08 AT %MX25544.8 : BOOL;
	bArm1VertStn11Down_09 AT %MX25544.9 : BOOL;
	bArm1VertStn11Down_10 AT %MX25544.10 : BOOL;
	bArm1VertStn11Down_11 AT %MX25544.11 : BOOL;
	bArm1VertStn11Down_12 AT %MX25544.12 : BOOL;
	bArm1VertStn11Down_13 AT %MX25544.13 : BOOL;
	bArm1VertStn11Down_14 AT %MX25544.14 : BOOL;
	bArm1VertStn11Down_15 AT %MX25544.15 : BOOL;
	bArm1VertStn11Down_16 AT %MX25544.16 : BOOL;
	bArm1VertStn11Down_17 AT %MX25544.17 : BOOL;
	bArm1VertStn11Down_18 AT %MX25544.18 : BOOL;
	bArm1VertStn11Down_19 AT %MX25544.19 : BOOL;
	bArm1VertStn11Down_20 AT %MX25544.20 : BOOL;
	bArm1VertStn11Down_21 AT %MX25544.21 : BOOL;
	bArm1VertStn11Down_22 AT %MX25544.22 : BOOL;
	bArm1VertStn11Down_23 AT %MX25544.23 : BOOL;
	bArm1VertStn11Down_24 AT %MX25544.24 : BOOL;
	bArm1VertStn11Down_25 AT %MX25544.25 : BOOL;
	bArm1VertStn11Down_26 AT %MX25544.26 : BOOL;
	bArm1VertStn11Down_27 AT %MX25544.27 : BOOL;
	bArm1VertStn11Down_28 AT %MX25544.28 : BOOL;
	bArm1VertStn11Down_29 AT %MX25544.29 : BOOL;
	bArm1VertStn11Down_30 AT %MX25544.30 : BOOL;
	bArm1VertStn11Down_31 AT %MX25544.31 : BOOL;

	bArm1VertStn12Down_00 AT %MX25548.0 : BOOL;
	bArm1VertStn12Down_01 AT %MX25548.1 : BOOL;
	bArm1VertStn12Down_02 AT %MX25548.2 : BOOL;
	bArm1VertStn12Down_03 AT %MX25548.3 : BOOL;
	bArm1VertStn12Down_04 AT %MX25548.4 : BOOL;
	bArm1VertStn12Down_05 AT %MX25548.5 : BOOL;
	bArm1VertStn12Down_06 AT %MX25548.6 : BOOL;
	bArm1VertStn12Down_07 AT %MX25548.7 : BOOL;
	bArm1VertStn12Down_08 AT %MX25548.8 : BOOL;
	bArm1VertStn12Down_09 AT %MX25548.9 : BOOL;
	bArm1VertStn12Down_10 AT %MX25548.10 : BOOL;
	bArm1VertStn12Down_11 AT %MX25548.11 : BOOL;
	bArm1VertStn12Down_12 AT %MX25548.12 : BOOL;
	bArm1VertStn12Down_13 AT %MX25548.13 : BOOL;
	bArm1VertStn12Down_14 AT %MX25548.14 : BOOL;
	bArm1VertStn12Down_15 AT %MX25548.15 : BOOL;
	bArm1VertStn12Down_16 AT %MX25548.16 : BOOL;
	bArm1VertStn12Down_17 AT %MX25548.17 : BOOL;
	bArm1VertStn12Down_18 AT %MX25548.18 : BOOL;
	bArm1VertStn12Down_19 AT %MX25548.19 : BOOL;
	bArm1VertStn12Down_20 AT %MX25548.20 : BOOL;
	bArm1VertStn12Down_21 AT %MX25548.21 : BOOL;
	bArm1VertStn12Down_22 AT %MX25548.22 : BOOL;
	bArm1VertStn12Down_23 AT %MX25548.23 : BOOL;
	bArm1VertStn12Down_24 AT %MX25548.24 : BOOL;
	bArm1VertStn12Down_25 AT %MX25548.25 : BOOL;
	bArm1VertStn12Down_26 AT %MX25548.26 : BOOL;
	bArm1VertStn12Down_27 AT %MX25548.27 : BOOL;
	bArm1VertStn12Down_28 AT %MX25548.28 : BOOL;
	bArm1VertStn12Down_29 AT %MX25548.29 : BOOL;
	bArm1VertStn12Down_30 AT %MX25548.30 : BOOL;
	bArm1VertStn12Down_31 AT %MX25548.31 : BOOL;


(* xxxxxxxxxxxxxxxxxxxxxxxxxxxxxxxxxxxxxxx Lifter xxxxxxxxxxxxxxxxxxxxxxxxxxxxxxxxxxxxxxx*)
(*========= Up/Down LifterUp BOOL LINK with %MX30000-  =========*)

	bSlowPull1LifterStn1Up_00 AT %MX30004.0 : BOOL;
	bSlowPull1LifterStn1Up_01 AT %MX30004.1 : BOOL;
	bSlowPull1LifterStn1Up_02 AT %MX30004.2 : BOOL;
	bSlowPull1LifterStn1Up_03 AT %MX30004.3 : BOOL;
	bSlowPull1LifterStn1Up_04 AT %MX30004.4 : BOOL;
	bSlowPull1LifterStn1Up_05 AT %MX30004.5 : BOOL;
	bSlowPull1LifterStn1Up_06 AT %MX30004.6 : BOOL;
	bSlowPull1LifterStn1Up_07 AT %MX30004.7 : BOOL;
	bSlowPull1LifterStn1Up_08 AT %MX30004.8 : BOOL;
	bSlowPull1LifterStn1Up_09 AT %MX30004.9 : BOOL;
	bSlowPull1LifterStn1Up_10 AT %MX30004.10 : BOOL;
	bSlowPull1LifterStn1Up_11 AT %MX30004.11 : BOOL;
	bSlowPull1LifterStn1Up_12 AT %MX30004.12 : BOOL;
	bSlowPull1LifterStn1Up_13 AT %MX30004.13 : BOOL;
	bSlowPull1LifterStn1Up_14 AT %MX30004.14 : BOOL;
	bSlowPull1LifterStn1Up_15 AT %MX30004.15 : BOOL;
	bSlowPull1LifterStn1Up_16 AT %MX30004.16 : BOOL;
	bSlowPull1LifterStn1Up_17 AT %MX30004.17 : BOOL;
	bSlowPull1LifterStn1Up_18 AT %MX30004.18 : BOOL;
	bSlowPull1LifterStn1Up_19 AT %MX30004.19 : BOOL;
	bSlowPull1LifterStn1Up_20 AT %MX30004.20 : BOOL;
	bSlowPull1LifterStn1Up_21 AT %MX30004.21 : BOOL;
	bSlowPull1LifterStn1Up_22 AT %MX30004.22 : BOOL;
	bSlowPull1LifterStn1Up_23 AT %MX30004.23 : BOOL;
	bSlowPull1LifterStn1Up_24 AT %MX30004.24 : BOOL;
	bSlowPull1LifterStn1Up_25 AT %MX30004.25 : BOOL;
	bSlowPull1LifterStn1Up_26 AT %MX30004.26 : BOOL;
	bSlowPull1LifterStn1Up_27 AT %MX30004.27 : BOOL;
	bSlowPull1LifterStn1Up_28 AT %MX30004.28 : BOOL;
	bSlowPull1LifterStn1Up_29 AT %MX30004.29 : BOOL;
	bSlowPull1LifterStn1Up_30 AT %MX30004.30 : BOOL;
	bSlowPull1LifterStn1Up_31 AT %MX30004.31 : BOOL;

	bSlowPull1LifterStn2Up_00 AT %MX30008.0 : BOOL;
	bSlowPull1LifterStn2Up_01 AT %MX30008.1 : BOOL;
	bSlowPull1LifterStn2Up_02 AT %MX30008.2 : BOOL;
	bSlowPull1LifterStn2Up_03 AT %MX30008.3 : BOOL;
	bSlowPull1LifterStn2Up_04 AT %MX30008.4 : BOOL;
	bSlowPull1LifterStn2Up_05 AT %MX30008.5 : BOOL;
	bSlowPull1LifterStn2Up_06 AT %MX30008.6 : BOOL;
	bSlowPull1LifterStn2Up_07 AT %MX30008.7 : BOOL;
	bSlowPull1LifterStn2Up_08 AT %MX30008.8 : BOOL;
	bSlowPull1LifterStn2Up_09 AT %MX30008.9 : BOOL;
	bSlowPull1LifterStn2Up_10 AT %MX30008.10 : BOOL;
	bSlowPull1LifterStn2Up_11 AT %MX30008.11 : BOOL;
	bSlowPull1LifterStn2Up_12 AT %MX30008.12 : BOOL;
	bSlowPull1LifterStn2Up_13 AT %MX30008.13 : BOOL;
	bSlowPull1LifterStn2Up_14 AT %MX30008.14 : BOOL;
	bSlowPull1LifterStn2Up_15 AT %MX30008.15 : BOOL;
	bSlowPull1LifterStn2Up_16 AT %MX30008.16 : BOOL;
	bSlowPull1LifterStn2Up_17 AT %MX30008.17 : BOOL;
	bSlowPull1LifterStn2Up_18 AT %MX30008.18 : BOOL;
	bSlowPull1LifterStn2Up_19 AT %MX30008.19 : BOOL;
	bSlowPull1LifterStn2Up_20 AT %MX30008.20 : BOOL;
	bSlowPull1LifterStn2Up_21 AT %MX30008.21 : BOOL;
	bSlowPull1LifterStn2Up_22 AT %MX30008.22 : BOOL;
	bSlowPull1LifterStn2Up_23 AT %MX30008.23 : BOOL;
	bSlowPull1LifterStn2Up_24 AT %MX30008.24 : BOOL;
	bSlowPull1LifterStn2Up_25 AT %MX30008.25 : BOOL;
	bSlowPull1LifterStn2Up_26 AT %MX30008.26 : BOOL;
	bSlowPull1LifterStn2Up_27 AT %MX30008.27 : BOOL;
	bSlowPull1LifterStn2Up_28 AT %MX30008.28 : BOOL;
	bSlowPull1LifterStn2Up_29 AT %MX30008.29 : BOOL;
	bSlowPull1LifterStn2Up_30 AT %MX30008.30 : BOOL;
	bSlowPull1LifterStn2Up_31 AT %MX30008.31 : BOOL;

	bSlowPull1LifterStn3Up_00 AT %MX30012.0 : BOOL;
	bSlowPull1LifterStn3Up_01 AT %MX30012.1 : BOOL;
	bSlowPull1LifterStn3Up_02 AT %MX30012.2 : BOOL;
	bSlowPull1LifterStn3Up_03 AT %MX30012.3 : BOOL;
	bSlowPull1LifterStn3Up_04 AT %MX30012.4 : BOOL;
	bSlowPull1LifterStn3Up_05 AT %MX30012.5 : BOOL;
	bSlowPull1LifterStn3Up_06 AT %MX30012.6 : BOOL;
	bSlowPull1LifterStn3Up_07 AT %MX30012.7 : BOOL;
	bSlowPull1LifterStn3Up_08 AT %MX30012.8 : BOOL;
	bSlowPull1LifterStn3Up_09 AT %MX30012.9 : BOOL;
	bSlowPull1LifterStn3Up_10 AT %MX30012.10 : BOOL;
	bSlowPull1LifterStn3Up_11 AT %MX30012.11 : BOOL;
	bSlowPull1LifterStn3Up_12 AT %MX30012.12 : BOOL;
	bSlowPull1LifterStn3Up_13 AT %MX30012.13 : BOOL;
	bSlowPull1LifterStn3Up_14 AT %MX30012.14 : BOOL;
	bSlowPull1LifterStn3Up_15 AT %MX30012.15 : BOOL;
	bSlowPull1LifterStn3Up_16 AT %MX30012.16 : BOOL;
	bSlowPull1LifterStn3Up_17 AT %MX30012.17 : BOOL;
	bSlowPull1LifterStn3Up_18 AT %MX30012.18 : BOOL;
	bSlowPull1LifterStn3Up_19 AT %MX30012.19 : BOOL;
	bSlowPull1LifterStn3Up_20 AT %MX30012.20 : BOOL;
	bSlowPull1LifterStn3Up_21 AT %MX30012.21 : BOOL;
	bSlowPull1LifterStn3Up_22 AT %MX30012.22 : BOOL;
	bSlowPull1LifterStn3Up_23 AT %MX30012.23 : BOOL;
	bSlowPull1LifterStn3Up_24 AT %MX30012.24 : BOOL;
	bSlowPull1LifterStn3Up_25 AT %MX30012.25 : BOOL;
	bSlowPull1LifterStn3Up_26 AT %MX30012.26 : BOOL;
	bSlowPull1LifterStn3Up_27 AT %MX30012.27 : BOOL;
	bSlowPull1LifterStn3Up_28 AT %MX30012.28 : BOOL;
	bSlowPull1LifterStn3Up_29 AT %MX30012.29 : BOOL;
	bSlowPull1LifterStn3Up_30 AT %MX30012.30 : BOOL;
	bSlowPull1LifterStn3Up_31 AT %MX30012.31 : BOOL;

	bSlowPull1LifterStn4Up_00 AT %MX30016.0 : BOOL;
	bSlowPull1LifterStn4Up_01 AT %MX30016.1 : BOOL;
	bSlowPull1LifterStn4Up_02 AT %MX30016.2 : BOOL;
	bSlowPull1LifterStn4Up_03 AT %MX30016.3 : BOOL;
	bSlowPull1LifterStn4Up_04 AT %MX30016.4 : BOOL;
	bSlowPull1LifterStn4Up_05 AT %MX30016.5 : BOOL;
	bSlowPull1LifterStn4Up_06 AT %MX30016.6 : BOOL;
	bSlowPull1LifterStn4Up_07 AT %MX30016.7 : BOOL;
	bSlowPull1LifterStn4Up_08 AT %MX30016.8 : BOOL;
	bSlowPull1LifterStn4Up_09 AT %MX30016.9 : BOOL;
	bSlowPull1LifterStn4Up_10 AT %MX30016.10 : BOOL;
	bSlowPull1LifterStn4Up_11 AT %MX30016.11 : BOOL;
	bSlowPull1LifterStn4Up_12 AT %MX30016.12 : BOOL;
	bSlowPull1LifterStn4Up_13 AT %MX30016.13 : BOOL;
	bSlowPull1LifterStn4Up_14 AT %MX30016.14 : BOOL;
	bSlowPull1LifterStn4Up_15 AT %MX30016.15 : BOOL;
	bSlowPull1LifterStn4Up_16 AT %MX30016.16 : BOOL;
	bSlowPull1LifterStn4Up_17 AT %MX30016.17 : BOOL;
	bSlowPull1LifterStn4Up_18 AT %MX30016.18 : BOOL;
	bSlowPull1LifterStn4Up_19 AT %MX30016.19 : BOOL;
	bSlowPull1LifterStn4Up_20 AT %MX30016.20 : BOOL;
	bSlowPull1LifterStn4Up_21 AT %MX30016.21 : BOOL;
	bSlowPull1LifterStn4Up_22 AT %MX30016.22 : BOOL;
	bSlowPull1LifterStn4Up_23 AT %MX30016.23 : BOOL;
	bSlowPull1LifterStn4Up_24 AT %MX30016.24 : BOOL;
	bSlowPull1LifterStn4Up_25 AT %MX30016.25 : BOOL;
	bSlowPull1LifterStn4Up_26 AT %MX30016.26 : BOOL;
	bSlowPull1LifterStn4Up_27 AT %MX30016.27 : BOOL;
	bSlowPull1LifterStn4Up_28 AT %MX30016.28 : BOOL;
	bSlowPull1LifterStn4Up_29 AT %MX30016.29 : BOOL;
	bSlowPull1LifterStn4Up_30 AT %MX30016.30 : BOOL;
	bSlowPull1LifterStn4Up_31 AT %MX30016.31 : BOOL;

	bSlowPull1LifterStn5Up_00 AT %MX30020.0 : BOOL;
	bSlowPull1LifterStn5Up_01 AT %MX30020.1 : BOOL;
	bSlowPull1LifterStn5Up_02 AT %MX30020.2 : BOOL;
	bSlowPull1LifterStn5Up_03 AT %MX30020.3 : BOOL;
	bSlowPull1LifterStn5Up_04 AT %MX30020.4 : BOOL;
	bSlowPull1LifterStn5Up_05 AT %MX30020.5 : BOOL;
	bSlowPull1LifterStn5Up_06 AT %MX30020.6 : BOOL;
	bSlowPull1LifterStn5Up_07 AT %MX30020.7 : BOOL;
	bSlowPull1LifterStn5Up_08 AT %MX30020.8 : BOOL;
	bSlowPull1LifterStn5Up_09 AT %MX30020.9 : BOOL;
	bSlowPull1LifterStn5Up_10 AT %MX30020.10 : BOOL;
	bSlowPull1LifterStn5Up_11 AT %MX30020.11 : BOOL;
	bSlowPull1LifterStn5Up_12 AT %MX30020.12 : BOOL;
	bSlowPull1LifterStn5Up_13 AT %MX30020.13 : BOOL;
	bSlowPull1LifterStn5Up_14 AT %MX30020.14 : BOOL;
	bSlowPull1LifterStn5Up_15 AT %MX30020.15 : BOOL;
	bSlowPull1LifterStn5Up_16 AT %MX30020.16 : BOOL;
	bSlowPull1LifterStn5Up_17 AT %MX30020.17 : BOOL;
	bSlowPull1LifterStn5Up_18 AT %MX30020.18 : BOOL;
	bSlowPull1LifterStn5Up_19 AT %MX30020.19 : BOOL;
	bSlowPull1LifterStn5Up_20 AT %MX30020.20 : BOOL;
	bSlowPull1LifterStn5Up_21 AT %MX30020.21 : BOOL;
	bSlowPull1LifterStn5Up_22 AT %MX30020.22 : BOOL;
	bSlowPull1LifterStn5Up_23 AT %MX30020.23 : BOOL;
	bSlowPull1LifterStn5Up_24 AT %MX30020.24 : BOOL;
	bSlowPull1LifterStn5Up_25 AT %MX30020.25 : BOOL;
	bSlowPull1LifterStn5Up_26 AT %MX30020.26 : BOOL;
	bSlowPull1LifterStn5Up_27 AT %MX30020.27 : BOOL;
	bSlowPull1LifterStn5Up_28 AT %MX30020.28 : BOOL;
	bSlowPull1LifterStn5Up_29 AT %MX30020.29 : BOOL;
	bSlowPull1LifterStn5Up_30 AT %MX30020.30 : BOOL;
	bSlowPull1LifterStn5Up_31 AT %MX30020.31 : BOOL;

	bSlowPull1LifterStn6Up_00 AT %MX30024.0 : BOOL;
	bSlowPull1LifterStn6Up_01 AT %MX30024.1 : BOOL;
	bSlowPull1LifterStn6Up_02 AT %MX30024.2 : BOOL;
	bSlowPull1LifterStn6Up_03 AT %MX30024.3 : BOOL;
	bSlowPull1LifterStn6Up_04 AT %MX30024.4 : BOOL;
	bSlowPull1LifterStn6Up_05 AT %MX30024.5 : BOOL;
	bSlowPull1LifterStn6Up_06 AT %MX30024.6 : BOOL;
	bSlowPull1LifterStn6Up_07 AT %MX30024.7 : BOOL;
	bSlowPull1LifterStn6Up_08 AT %MX30024.8 : BOOL;
	bSlowPull1LifterStn6Up_09 AT %MX30024.9 : BOOL;
	bSlowPull1LifterStn6Up_10 AT %MX30024.10 : BOOL;
	bSlowPull1LifterStn6Up_11 AT %MX30024.11 : BOOL;
	bSlowPull1LifterStn6Up_12 AT %MX30024.12 : BOOL;
	bSlowPull1LifterStn6Up_13 AT %MX30024.13 : BOOL;
	bSlowPull1LifterStn6Up_14 AT %MX30024.14 : BOOL;
	bSlowPull1LifterStn6Up_15 AT %MX30024.15 : BOOL;
	bSlowPull1LifterStn6Up_16 AT %MX30024.16 : BOOL;
	bSlowPull1LifterStn6Up_17 AT %MX30024.17 : BOOL;
	bSlowPull1LifterStn6Up_18 AT %MX30024.18 : BOOL;
	bSlowPull1LifterStn6Up_19 AT %MX30024.19 : BOOL;
	bSlowPull1LifterStn6Up_20 AT %MX30024.20 : BOOL;
	bSlowPull1LifterStn6Up_21 AT %MX30024.21 : BOOL;
	bSlowPull1LifterStn6Up_22 AT %MX30024.22 : BOOL;
	bSlowPull1LifterStn6Up_23 AT %MX30024.23 : BOOL;
	bSlowPull1LifterStn6Up_24 AT %MX30024.24 : BOOL;
	bSlowPull1LifterStn6Up_25 AT %MX30024.25 : BOOL;
	bSlowPull1LifterStn6Up_26 AT %MX30024.26 : BOOL;
	bSlowPull1LifterStn6Up_27 AT %MX30024.27 : BOOL;
	bSlowPull1LifterStn6Up_28 AT %MX30024.28 : BOOL;
	bSlowPull1LifterStn6Up_29 AT %MX30024.29 : BOOL;
	bSlowPull1LifterStn6Up_30 AT %MX30024.30 : BOOL;
	bSlowPull1LifterStn6Up_31 AT %MX30024.31 : BOOL;

	bSlowPull1LifterStn7Up_00 AT %MX30028.0 : BOOL;
	bSlowPull1LifterStn7Up_01 AT %MX30028.1 : BOOL;
	bSlowPull1LifterStn7Up_02 AT %MX30028.2 : BOOL;
	bSlowPull1LifterStn7Up_03 AT %MX30028.3 : BOOL;
	bSlowPull1LifterStn7Up_04 AT %MX30028.4 : BOOL;
	bSlowPull1LifterStn7Up_05 AT %MX30028.5 : BOOL;
	bSlowPull1LifterStn7Up_06 AT %MX30028.6 : BOOL;
	bSlowPull1LifterStn7Up_07 AT %MX30028.7 : BOOL;
	bSlowPull1LifterStn7Up_08 AT %MX30028.8 : BOOL;
	bSlowPull1LifterStn7Up_09 AT %MX30028.9 : BOOL;
	bSlowPull1LifterStn7Up_10 AT %MX30028.10 : BOOL;
	bSlowPull1LifterStn7Up_11 AT %MX30028.11 : BOOL;
	bSlowPull1LifterStn7Up_12 AT %MX30028.12 : BOOL;
	bSlowPull1LifterStn7Up_13 AT %MX30028.13 : BOOL;
	bSlowPull1LifterStn7Up_14 AT %MX30028.14 : BOOL;
	bSlowPull1LifterStn7Up_15 AT %MX30028.15 : BOOL;
	bSlowPull1LifterStn7Up_16 AT %MX30028.16 : BOOL;
	bSlowPull1LifterStn7Up_17 AT %MX30028.17 : BOOL;
	bSlowPull1LifterStn7Up_18 AT %MX30028.18 : BOOL;
	bSlowPull1LifterStn7Up_19 AT %MX30028.19 : BOOL;
	bSlowPull1LifterStn7Up_20 AT %MX30028.20 : BOOL;
	bSlowPull1LifterStn7Up_21 AT %MX30028.21 : BOOL;
	bSlowPull1LifterStn7Up_22 AT %MX30028.22 : BOOL;
	bSlowPull1LifterStn7Up_23 AT %MX30028.23 : BOOL;
	bSlowPull1LifterStn7Up_24 AT %MX30028.24 : BOOL;
	bSlowPull1LifterStn7Up_25 AT %MX30028.25 : BOOL;
	bSlowPull1LifterStn7Up_26 AT %MX30028.26 : BOOL;
	bSlowPull1LifterStn7Up_27 AT %MX30028.27 : BOOL;
	bSlowPull1LifterStn7Up_28 AT %MX30028.28 : BOOL;
	bSlowPull1LifterStn7Up_29 AT %MX30028.29 : BOOL;
	bSlowPull1LifterStn7Up_30 AT %MX30028.30 : BOOL;
	bSlowPull1LifterStn7Up_31 AT %MX30028.31 : BOOL;

	bSlowPull1LifterStn8Up_00 AT %MX30032.0 : BOOL;
	bSlowPull1LifterStn8Up_01 AT %MX30032.1 : BOOL;
	bSlowPull1LifterStn8Up_02 AT %MX30032.2 : BOOL;
	bSlowPull1LifterStn8Up_03 AT %MX30032.3 : BOOL;
	bSlowPull1LifterStn8Up_04 AT %MX30032.4 : BOOL;
	bSlowPull1LifterStn8Up_05 AT %MX30032.5 : BOOL;
	bSlowPull1LifterStn8Up_06 AT %MX30032.6 : BOOL;
	bSlowPull1LifterStn8Up_07 AT %MX30032.7 : BOOL;
	bSlowPull1LifterStn8Up_08 AT %MX30032.8 : BOOL;
	bSlowPull1LifterStn8Up_09 AT %MX30032.9 : BOOL;
	bSlowPull1LifterStn8Up_10 AT %MX30032.10 : BOOL;
	bSlowPull1LifterStn8Up_11 AT %MX30032.11 : BOOL;
	bSlowPull1LifterStn8Up_12 AT %MX30032.12 : BOOL;
	bSlowPull1LifterStn8Up_13 AT %MX30032.13 : BOOL;
	bSlowPull1LifterStn8Up_14 AT %MX30032.14 : BOOL;
	bSlowPull1LifterStn8Up_15 AT %MX30032.15 : BOOL;
	bSlowPull1LifterStn8Up_16 AT %MX30032.16 : BOOL;
	bSlowPull1LifterStn8Up_17 AT %MX30032.17 : BOOL;
	bSlowPull1LifterStn8Up_18 AT %MX30032.18 : BOOL;
	bSlowPull1LifterStn8Up_19 AT %MX30032.19 : BOOL;
	bSlowPull1LifterStn8Up_20 AT %MX30032.20 : BOOL;
	bSlowPull1LifterStn8Up_21 AT %MX30032.21 : BOOL;
	bSlowPull1LifterStn8Up_22 AT %MX30032.22 : BOOL;
	bSlowPull1LifterStn8Up_23 AT %MX30032.23 : BOOL;
	bSlowPull1LifterStn8Up_24 AT %MX30032.24 : BOOL;
	bSlowPull1LifterStn8Up_25 AT %MX30032.25 : BOOL;
	bSlowPull1LifterStn8Up_26 AT %MX30032.26 : BOOL;
	bSlowPull1LifterStn8Up_27 AT %MX30032.27 : BOOL;
	bSlowPull1LifterStn8Up_28 AT %MX30032.28 : BOOL;
	bSlowPull1LifterStn8Up_29 AT %MX30032.29 : BOOL;
	bSlowPull1LifterStn8Up_30 AT %MX30032.30 : BOOL;
	bSlowPull1LifterStn8Up_31 AT %MX30032.31 : BOOL;

	bSlowPull1LifterStn9Up_00 AT %MX30036.0 : BOOL;
	bSlowPull1LifterStn9Up_01 AT %MX30036.1 : BOOL;
	bSlowPull1LifterStn9Up_02 AT %MX30036.2 : BOOL;
	bSlowPull1LifterStn9Up_03 AT %MX30036.3 : BOOL;
	bSlowPull1LifterStn9Up_04 AT %MX30036.4 : BOOL;
	bSlowPull1LifterStn9Up_05 AT %MX30036.5 : BOOL;
	bSlowPull1LifterStn9Up_06 AT %MX30036.6 : BOOL;
	bSlowPull1LifterStn9Up_07 AT %MX30036.7 : BOOL;
	bSlowPull1LifterStn9Up_08 AT %MX30036.8 : BOOL;
	bSlowPull1LifterStn9Up_09 AT %MX30036.9 : BOOL;
	bSlowPull1LifterStn9Up_10 AT %MX30036.10 : BOOL;
	bSlowPull1LifterStn9Up_11 AT %MX30036.11 : BOOL;
	bSlowPull1LifterStn9Up_12 AT %MX30036.12 : BOOL;
	bSlowPull1LifterStn9Up_13 AT %MX30036.13 : BOOL;
	bSlowPull1LifterStn9Up_14 AT %MX30036.14 : BOOL;
	bSlowPull1LifterStn9Up_15 AT %MX30036.15 : BOOL;
	bSlowPull1LifterStn9Up_16 AT %MX30036.16 : BOOL;
	bSlowPull1LifterStn9Up_17 AT %MX30036.17 : BOOL;
	bSlowPull1LifterStn9Up_18 AT %MX30036.18 : BOOL;
	bSlowPull1LifterStn9Up_19 AT %MX30036.19 : BOOL;
	bSlowPull1LifterStn9Up_20 AT %MX30036.20 : BOOL;
	bSlowPull1LifterStn9Up_21 AT %MX30036.21 : BOOL;
	bSlowPull1LifterStn9Up_22 AT %MX30036.22 : BOOL;
	bSlowPull1LifterStn9Up_23 AT %MX30036.23 : BOOL;
	bSlowPull1LifterStn9Up_24 AT %MX30036.24 : BOOL;
	bSlowPull1LifterStn9Up_25 AT %MX30036.25 : BOOL;
	bSlowPull1LifterStn9Up_26 AT %MX30036.26 : BOOL;
	bSlowPull1LifterStn9Up_27 AT %MX30036.27 : BOOL;
	bSlowPull1LifterStn9Up_28 AT %MX30036.28 : BOOL;
	bSlowPull1LifterStn9Up_29 AT %MX30036.29 : BOOL;
	bSlowPull1LifterStn9Up_30 AT %MX30036.30 : BOOL;
	bSlowPull1LifterStn9Up_31 AT %MX30036.31 : BOOL;

	bSlowPull1LifterStn10Up_00 AT %MX30040.0 : BOOL;
	bSlowPull1LifterStn10Up_01 AT %MX30040.1 : BOOL;
	bSlowPull1LifterStn10Up_02 AT %MX30040.2 : BOOL;
	bSlowPull1LifterStn10Up_03 AT %MX30040.3 : BOOL;
	bSlowPull1LifterStn10Up_04 AT %MX30040.4 : BOOL;
	bSlowPull1LifterStn10Up_05 AT %MX30040.5 : BOOL;
	bSlowPull1LifterStn10Up_06 AT %MX30040.6 : BOOL;
	bSlowPull1LifterStn10Up_07 AT %MX30040.7 : BOOL;
	bSlowPull1LifterStn10Up_08 AT %MX30040.8 : BOOL;
	bSlowPull1LifterStn10Up_09 AT %MX30040.9 : BOOL;
	bSlowPull1LifterStn10Up_10 AT %MX30040.10 : BOOL;
	bSlowPull1LifterStn10Up_11 AT %MX30040.11 : BOOL;
	bSlowPull1LifterStn10Up_12 AT %MX30040.12 : BOOL;
	bSlowPull1LifterStn10Up_13 AT %MX30040.13 : BOOL;
	bSlowPull1LifterStn10Up_14 AT %MX30040.14 : BOOL;
	bSlowPull1LifterStn10Up_15 AT %MX30040.15 : BOOL;
	bSlowPull1LifterStn10Up_16 AT %MX30040.16 : BOOL;
	bSlowPull1LifterStn10Up_17 AT %MX30040.17 : BOOL;
	bSlowPull1LifterStn10Up_18 AT %MX30040.18 : BOOL;
	bSlowPull1LifterStn10Up_19 AT %MX30040.19 : BOOL;
	bSlowPull1LifterStn10Up_20 AT %MX30040.20 : BOOL;
	bSlowPull1LifterStn10Up_21 AT %MX30040.21 : BOOL;
	bSlowPull1LifterStn10Up_22 AT %MX30040.22 : BOOL;
	bSlowPull1LifterStn10Up_23 AT %MX30040.23 : BOOL;
	bSlowPull1LifterStn10Up_24 AT %MX30040.24 : BOOL;
	bSlowPull1LifterStn10Up_25 AT %MX30040.25 : BOOL;
	bSlowPull1LifterStn10Up_26 AT %MX30040.26 : BOOL;
	bSlowPull1LifterStn10Up_27 AT %MX30040.27 : BOOL;
	bSlowPull1LifterStn10Up_28 AT %MX30040.28 : BOOL;
	bSlowPull1LifterStn10Up_29 AT %MX30040.29 : BOOL;
	bSlowPull1LifterStn10Up_30 AT %MX30040.30 : BOOL;
	bSlowPull1LifterStn10Up_31 AT %MX30040.31 : BOOL;


(* xxxxxxxxxxxxxxxxxxxxxxxxxxxxxxxxxxxxxxx Lifter xxxxxxxxxxxxxxxxxxxxxxxxxxxxxxxxxxxxxxx*)
(*========= Up/Down LifterDown BOOL LINK with %MX30000-  =========*)

	bSlowPull1LifterStn1Down_00 AT %MX30304.0 : BOOL;
	bSlowPull1LifterStn1Down_01 AT %MX30304.1 : BOOL;
	bSlowPull1LifterStn1Down_02 AT %MX30304.2 : BOOL;
	bSlowPull1LifterStn1Down_03 AT %MX30304.3 : BOOL;
	bSlowPull1LifterStn1Down_04 AT %MX30304.4 : BOOL;
	bSlowPull1LifterStn1Down_05 AT %MX30304.5 : BOOL;
	bSlowPull1LifterStn1Down_06 AT %MX30304.6 : BOOL;
	bSlowPull1LifterStn1Down_07 AT %MX30304.7 : BOOL;
	bSlowPull1LifterStn1Down_08 AT %MX30304.8 : BOOL;
	bSlowPull1LifterStn1Down_09 AT %MX30304.9 : BOOL;
	bSlowPull1LifterStn1Down_10 AT %MX30304.10 : BOOL;
	bSlowPull1LifterStn1Down_11 AT %MX30304.11 : BOOL;
	bSlowPull1LifterStn1Down_12 AT %MX30304.12 : BOOL;
	bSlowPull1LifterStn1Down_13 AT %MX30304.13 : BOOL;
	bSlowPull1LifterStn1Down_14 AT %MX30304.14 : BOOL;
	bSlowPull1LifterStn1Down_15 AT %MX30304.15 : BOOL;
	bSlowPull1LifterStn1Down_16 AT %MX30304.16 : BOOL;
	bSlowPull1LifterStn1Down_17 AT %MX30304.17 : BOOL;
	bSlowPull1LifterStn1Down_18 AT %MX30304.18 : BOOL;
	bSlowPull1LifterStn1Down_19 AT %MX30304.19 : BOOL;
	bSlowPull1LifterStn1Down_20 AT %MX30304.20 : BOOL;
	bSlowPull1LifterStn1Down_21 AT %MX30304.21 : BOOL;
	bSlowPull1LifterStn1Down_22 AT %MX30304.22 : BOOL;
	bSlowPull1LifterStn1Down_23 AT %MX30304.23 : BOOL;
	bSlowPull1LifterStn1Down_24 AT %MX30304.24 : BOOL;
	bSlowPull1LifterStn1Down_25 AT %MX30304.25 : BOOL;
	bSlowPull1LifterStn1Down_26 AT %MX30304.26 : BOOL;
	bSlowPull1LifterStn1Down_27 AT %MX30304.27 : BOOL;
	bSlowPull1LifterStn1Down_28 AT %MX30304.28 : BOOL;
	bSlowPull1LifterStn1Down_29 AT %MX30304.29 : BOOL;
	bSlowPull1LifterStn1Down_30 AT %MX30304.30 : BOOL;
	bSlowPull1LifterStn1Down_31 AT %MX30304.31 : BOOL;

	bSlowPull1LifterStn2Down_00 AT %MX30308.0 : BOOL;
	bSlowPull1LifterStn2Down_01 AT %MX30308.1 : BOOL;
	bSlowPull1LifterStn2Down_02 AT %MX30308.2 : BOOL;
	bSlowPull1LifterStn2Down_03 AT %MX30308.3 : BOOL;
	bSlowPull1LifterStn2Down_04 AT %MX30308.4 : BOOL;
	bSlowPull1LifterStn2Down_05 AT %MX30308.5 : BOOL;
	bSlowPull1LifterStn2Down_06 AT %MX30308.6 : BOOL;
	bSlowPull1LifterStn2Down_07 AT %MX30308.7 : BOOL;
	bSlowPull1LifterStn2Down_08 AT %MX30308.8 : BOOL;
	bSlowPull1LifterStn2Down_09 AT %MX30308.9 : BOOL;
	bSlowPull1LifterStn2Down_10 AT %MX30308.10 : BOOL;
	bSlowPull1LifterStn2Down_11 AT %MX30308.11 : BOOL;
	bSlowPull1LifterStn2Down_12 AT %MX30308.12 : BOOL;
	bSlowPull1LifterStn2Down_13 AT %MX30308.13 : BOOL;
	bSlowPull1LifterStn2Down_14 AT %MX30308.14 : BOOL;
	bSlowPull1LifterStn2Down_15 AT %MX30308.15 : BOOL;
	bSlowPull1LifterStn2Down_16 AT %MX30308.16 : BOOL;
	bSlowPull1LifterStn2Down_17 AT %MX30308.17 : BOOL;
	bSlowPull1LifterStn2Down_18 AT %MX30308.18 : BOOL;
	bSlowPull1LifterStn2Down_19 AT %MX30308.19 : BOOL;
	bSlowPull1LifterStn2Down_20 AT %MX30308.20 : BOOL;
	bSlowPull1LifterStn2Down_21 AT %MX30308.21 : BOOL;
	bSlowPull1LifterStn2Down_22 AT %MX30308.22 : BOOL;
	bSlowPull1LifterStn2Down_23 AT %MX30308.23 : BOOL;
	bSlowPull1LifterStn2Down_24 AT %MX30308.24 : BOOL;
	bSlowPull1LifterStn2Down_25 AT %MX30308.25 : BOOL;
	bSlowPull1LifterStn2Down_26 AT %MX30308.26 : BOOL;
	bSlowPull1LifterStn2Down_27 AT %MX30308.27 : BOOL;
	bSlowPull1LifterStn2Down_28 AT %MX30308.28 : BOOL;
	bSlowPull1LifterStn2Down_29 AT %MX30308.29 : BOOL;
	bSlowPull1LifterStn2Down_30 AT %MX30308.30 : BOOL;
	bSlowPull1LifterStn2Down_31 AT %MX30308.31 : BOOL;

	bSlowPull1LifterStn3Down_00 AT %MX30312.0 : BOOL;
	bSlowPull1LifterStn3Down_01 AT %MX30312.1 : BOOL;
	bSlowPull1LifterStn3Down_02 AT %MX30312.2 : BOOL;
	bSlowPull1LifterStn3Down_03 AT %MX30312.3 : BOOL;
	bSlowPull1LifterStn3Down_04 AT %MX30312.4 : BOOL;
	bSlowPull1LifterStn3Down_05 AT %MX30312.5 : BOOL;
	bSlowPull1LifterStn3Down_06 AT %MX30312.6 : BOOL;
	bSlowPull1LifterStn3Down_07 AT %MX30312.7 : BOOL;
	bSlowPull1LifterStn3Down_08 AT %MX30312.8 : BOOL;
	bSlowPull1LifterStn3Down_09 AT %MX30312.9 : BOOL;
	bSlowPull1LifterStn3Down_10 AT %MX30312.10 : BOOL;
	bSlowPull1LifterStn3Down_11 AT %MX30312.11 : BOOL;
	bSlowPull1LifterStn3Down_12 AT %MX30312.12 : BOOL;
	bSlowPull1LifterStn3Down_13 AT %MX30312.13 : BOOL;
	bSlowPull1LifterStn3Down_14 AT %MX30312.14 : BOOL;
	bSlowPull1LifterStn3Down_15 AT %MX30312.15 : BOOL;
	bSlowPull1LifterStn3Down_16 AT %MX30312.16 : BOOL;
	bSlowPull1LifterStn3Down_17 AT %MX30312.17 : BOOL;
	bSlowPull1LifterStn3Down_18 AT %MX30312.18 : BOOL;
	bSlowPull1LifterStn3Down_19 AT %MX30312.19 : BOOL;
	bSlowPull1LifterStn3Down_20 AT %MX30312.20 : BOOL;
	bSlowPull1LifterStn3Down_21 AT %MX30312.21 : BOOL;
	bSlowPull1LifterStn3Down_22 AT %MX30312.22 : BOOL;
	bSlowPull1LifterStn3Down_23 AT %MX30312.23 : BOOL;
	bSlowPull1LifterStn3Down_24 AT %MX30312.24 : BOOL;
	bSlowPull1LifterStn3Down_25 AT %MX30312.25 : BOOL;
	bSlowPull1LifterStn3Down_26 AT %MX30312.26 : BOOL;
	bSlowPull1LifterStn3Down_27 AT %MX30312.27 : BOOL;
	bSlowPull1LifterStn3Down_28 AT %MX30312.28 : BOOL;
	bSlowPull1LifterStn3Down_29 AT %MX30312.29 : BOOL;
	bSlowPull1LifterStn3Down_30 AT %MX30312.30 : BOOL;
	bSlowPull1LifterStn3Down_31 AT %MX30312.31 : BOOL;

	bSlowPull1LifterStn4Down_00 AT %MX30316.0 : BOOL;
	bSlowPull1LifterStn4Down_01 AT %MX30316.1 : BOOL;
	bSlowPull1LifterStn4Down_02 AT %MX30316.2 : BOOL;
	bSlowPull1LifterStn4Down_03 AT %MX30316.3 : BOOL;
	bSlowPull1LifterStn4Down_04 AT %MX30316.4 : BOOL;
	bSlowPull1LifterStn4Down_05 AT %MX30316.5 : BOOL;
	bSlowPull1LifterStn4Down_06 AT %MX30316.6 : BOOL;
	bSlowPull1LifterStn4Down_07 AT %MX30316.7 : BOOL;
	bSlowPull1LifterStn4Down_08 AT %MX30316.8 : BOOL;
	bSlowPull1LifterStn4Down_09 AT %MX30316.9 : BOOL;
	bSlowPull1LifterStn4Down_10 AT %MX30316.10 : BOOL;
	bSlowPull1LifterStn4Down_11 AT %MX30316.11 : BOOL;
	bSlowPull1LifterStn4Down_12 AT %MX30316.12 : BOOL;
	bSlowPull1LifterStn4Down_13 AT %MX30316.13 : BOOL;
	bSlowPull1LifterStn4Down_14 AT %MX30316.14 : BOOL;
	bSlowPull1LifterStn4Down_15 AT %MX30316.15 : BOOL;
	bSlowPull1LifterStn4Down_16 AT %MX30316.16 : BOOL;
	bSlowPull1LifterStn4Down_17 AT %MX30316.17 : BOOL;
	bSlowPull1LifterStn4Down_18 AT %MX30316.18 : BOOL;
	bSlowPull1LifterStn4Down_19 AT %MX30316.19 : BOOL;
	bSlowPull1LifterStn4Down_20 AT %MX30316.20 : BOOL;
	bSlowPull1LifterStn4Down_21 AT %MX30316.21 : BOOL;
	bSlowPull1LifterStn4Down_22 AT %MX30316.22 : BOOL;
	bSlowPull1LifterStn4Down_23 AT %MX30316.23 : BOOL;
	bSlowPull1LifterStn4Down_24 AT %MX30316.24 : BOOL;
	bSlowPull1LifterStn4Down_25 AT %MX30316.25 : BOOL;
	bSlowPull1LifterStn4Down_26 AT %MX30316.26 : BOOL;
	bSlowPull1LifterStn4Down_27 AT %MX30316.27 : BOOL;
	bSlowPull1LifterStn4Down_28 AT %MX30316.28 : BOOL;
	bSlowPull1LifterStn4Down_29 AT %MX30316.29 : BOOL;
	bSlowPull1LifterStn4Down_30 AT %MX30316.30 : BOOL;
	bSlowPull1LifterStn4Down_31 AT %MX30316.31 : BOOL;

	bSlowPull1LifterStn5Down_00 AT %MX30320.0 : BOOL;
	bSlowPull1LifterStn5Down_01 AT %MX30320.1 : BOOL;
	bSlowPull1LifterStn5Down_02 AT %MX30320.2 : BOOL;
	bSlowPull1LifterStn5Down_03 AT %MX30320.3 : BOOL;
	bSlowPull1LifterStn5Down_04 AT %MX30320.4 : BOOL;
	bSlowPull1LifterStn5Down_05 AT %MX30320.5 : BOOL;
	bSlowPull1LifterStn5Down_06 AT %MX30320.6 : BOOL;
	bSlowPull1LifterStn5Down_07 AT %MX30320.7 : BOOL;
	bSlowPull1LifterStn5Down_08 AT %MX30320.8 : BOOL;
	bSlowPull1LifterStn5Down_09 AT %MX30320.9 : BOOL;
	bSlowPull1LifterStn5Down_10 AT %MX30320.10 : BOOL;
	bSlowPull1LifterStn5Down_11 AT %MX30320.11 : BOOL;
	bSlowPull1LifterStn5Down_12 AT %MX30320.12 : BOOL;
	bSlowPull1LifterStn5Down_13 AT %MX30320.13 : BOOL;
	bSlowPull1LifterStn5Down_14 AT %MX30320.14 : BOOL;
	bSlowPull1LifterStn5Down_15 AT %MX30320.15 : BOOL;
	bSlowPull1LifterStn5Down_16 AT %MX30320.16 : BOOL;
	bSlowPull1LifterStn5Down_17 AT %MX30320.17 : BOOL;
	bSlowPull1LifterStn5Down_18 AT %MX30320.18 : BOOL;
	bSlowPull1LifterStn5Down_19 AT %MX30320.19 : BOOL;
	bSlowPull1LifterStn5Down_20 AT %MX30320.20 : BOOL;
	bSlowPull1LifterStn5Down_21 AT %MX30320.21 : BOOL;
	bSlowPull1LifterStn5Down_22 AT %MX30320.22 : BOOL;
	bSlowPull1LifterStn5Down_23 AT %MX30320.23 : BOOL;
	bSlowPull1LifterStn5Down_24 AT %MX30320.24 : BOOL;
	bSlowPull1LifterStn5Down_25 AT %MX30320.25 : BOOL;
	bSlowPull1LifterStn5Down_26 AT %MX30320.26 : BOOL;
	bSlowPull1LifterStn5Down_27 AT %MX30320.27 : BOOL;
	bSlowPull1LifterStn5Down_28 AT %MX30320.28 : BOOL;
	bSlowPull1LifterStn5Down_29 AT %MX30320.29 : BOOL;
	bSlowPull1LifterStn5Down_30 AT %MX30320.30 : BOOL;
	bSlowPull1LifterStn5Down_31 AT %MX30320.31 : BOOL;

	bSlowPull1LifterStn6Down_00 AT %MX30324.0 : BOOL;
	bSlowPull1LifterStn6Down_01 AT %MX30324.1 : BOOL;
	bSlowPull1LifterStn6Down_02 AT %MX30324.2 : BOOL;
	bSlowPull1LifterStn6Down_03 AT %MX30324.3 : BOOL;
	bSlowPull1LifterStn6Down_04 AT %MX30324.4 : BOOL;
	bSlowPull1LifterStn6Down_05 AT %MX30324.5 : BOOL;
	bSlowPull1LifterStn6Down_06 AT %MX30324.6 : BOOL;
	bSlowPull1LifterStn6Down_07 AT %MX30324.7 : BOOL;
	bSlowPull1LifterStn6Down_08 AT %MX30324.8 : BOOL;
	bSlowPull1LifterStn6Down_09 AT %MX30324.9 : BOOL;
	bSlowPull1LifterStn6Down_10 AT %MX30324.10 : BOOL;
	bSlowPull1LifterStn6Down_11 AT %MX30324.11 : BOOL;
	bSlowPull1LifterStn6Down_12 AT %MX30324.12 : BOOL;
	bSlowPull1LifterStn6Down_13 AT %MX30324.13 : BOOL;
	bSlowPull1LifterStn6Down_14 AT %MX30324.14 : BOOL;
	bSlowPull1LifterStn6Down_15 AT %MX30324.15 : BOOL;
	bSlowPull1LifterStn6Down_16 AT %MX30324.16 : BOOL;
	bSlowPull1LifterStn6Down_17 AT %MX30324.17 : BOOL;
	bSlowPull1LifterStn6Down_18 AT %MX30324.18 : BOOL;
	bSlowPull1LifterStn6Down_19 AT %MX30324.19 : BOOL;
	bSlowPull1LifterStn6Down_20 AT %MX30324.20 : BOOL;
	bSlowPull1LifterStn6Down_21 AT %MX30324.21 : BOOL;
	bSlowPull1LifterStn6Down_22 AT %MX30324.22 : BOOL;
	bSlowPull1LifterStn6Down_23 AT %MX30324.23 : BOOL;
	bSlowPull1LifterStn6Down_24 AT %MX30324.24 : BOOL;
	bSlowPull1LifterStn6Down_25 AT %MX30324.25 : BOOL;
	bSlowPull1LifterStn6Down_26 AT %MX30324.26 : BOOL;
	bSlowPull1LifterStn6Down_27 AT %MX30324.27 : BOOL;
	bSlowPull1LifterStn6Down_28 AT %MX30324.28 : BOOL;
	bSlowPull1LifterStn6Down_29 AT %MX30324.29 : BOOL;
	bSlowPull1LifterStn6Down_30 AT %MX30324.30 : BOOL;
	bSlowPull1LifterStn6Down_31 AT %MX30324.31 : BOOL;

	bSlowPull1LifterStn7Down_00 AT %MX30328.0 : BOOL;
	bSlowPull1LifterStn7Down_01 AT %MX30328.1 : BOOL;
	bSlowPull1LifterStn7Down_02 AT %MX30328.2 : BOOL;
	bSlowPull1LifterStn7Down_03 AT %MX30328.3 : BOOL;
	bSlowPull1LifterStn7Down_04 AT %MX30328.4 : BOOL;
	bSlowPull1LifterStn7Down_05 AT %MX30328.5 : BOOL;
	bSlowPull1LifterStn7Down_06 AT %MX30328.6 : BOOL;
	bSlowPull1LifterStn7Down_07 AT %MX30328.7 : BOOL;
	bSlowPull1LifterStn7Down_08 AT %MX30328.8 : BOOL;
	bSlowPull1LifterStn7Down_09 AT %MX30328.9 : BOOL;
	bSlowPull1LifterStn7Down_10 AT %MX30328.10 : BOOL;
	bSlowPull1LifterStn7Down_11 AT %MX30328.11 : BOOL;
	bSlowPull1LifterStn7Down_12 AT %MX30328.12 : BOOL;
	bSlowPull1LifterStn7Down_13 AT %MX30328.13 : BOOL;
	bSlowPull1LifterStn7Down_14 AT %MX30328.14 : BOOL;
	bSlowPull1LifterStn7Down_15 AT %MX30328.15 : BOOL;
	bSlowPull1LifterStn7Down_16 AT %MX30328.16 : BOOL;
	bSlowPull1LifterStn7Down_17 AT %MX30328.17 : BOOL;
	bSlowPull1LifterStn7Down_18 AT %MX30328.18 : BOOL;
	bSlowPull1LifterStn7Down_19 AT %MX30328.19 : BOOL;
	bSlowPull1LifterStn7Down_20 AT %MX30328.20 : BOOL;
	bSlowPull1LifterStn7Down_21 AT %MX30328.21 : BOOL;
	bSlowPull1LifterStn7Down_22 AT %MX30328.22 : BOOL;
	bSlowPull1LifterStn7Down_23 AT %MX30328.23 : BOOL;
	bSlowPull1LifterStn7Down_24 AT %MX30328.24 : BOOL;
	bSlowPull1LifterStn7Down_25 AT %MX30328.25 : BOOL;
	bSlowPull1LifterStn7Down_26 AT %MX30328.26 : BOOL;
	bSlowPull1LifterStn7Down_27 AT %MX30328.27 : BOOL;
	bSlowPull1LifterStn7Down_28 AT %MX30328.28 : BOOL;
	bSlowPull1LifterStn7Down_29 AT %MX30328.29 : BOOL;
	bSlowPull1LifterStn7Down_30 AT %MX30328.30 : BOOL;
	bSlowPull1LifterStn7Down_31 AT %MX30328.31 : BOOL;

	bSlowPull1LifterStn8Down_00 AT %MX30332.0 : BOOL;
	bSlowPull1LifterStn8Down_01 AT %MX30332.1 : BOOL;
	bSlowPull1LifterStn8Down_02 AT %MX30332.2 : BOOL;
	bSlowPull1LifterStn8Down_03 AT %MX30332.3 : BOOL;
	bSlowPull1LifterStn8Down_04 AT %MX30332.4 : BOOL;
	bSlowPull1LifterStn8Down_05 AT %MX30332.5 : BOOL;
	bSlowPull1LifterStn8Down_06 AT %MX30332.6 : BOOL;
	bSlowPull1LifterStn8Down_07 AT %MX30332.7 : BOOL;
	bSlowPull1LifterStn8Down_08 AT %MX30332.8 : BOOL;
	bSlowPull1LifterStn8Down_09 AT %MX30332.9 : BOOL;
	bSlowPull1LifterStn8Down_10 AT %MX30332.10 : BOOL;
	bSlowPull1LifterStn8Down_11 AT %MX30332.11 : BOOL;
	bSlowPull1LifterStn8Down_12 AT %MX30332.12 : BOOL;
	bSlowPull1LifterStn8Down_13 AT %MX30332.13 : BOOL;
	bSlowPull1LifterStn8Down_14 AT %MX30332.14 : BOOL;
	bSlowPull1LifterStn8Down_15 AT %MX30332.15 : BOOL;
	bSlowPull1LifterStn8Down_16 AT %MX30332.16 : BOOL;
	bSlowPull1LifterStn8Down_17 AT %MX30332.17 : BOOL;
	bSlowPull1LifterStn8Down_18 AT %MX30332.18 : BOOL;
	bSlowPull1LifterStn8Down_19 AT %MX30332.19 : BOOL;
	bSlowPull1LifterStn8Down_20 AT %MX30332.20 : BOOL;
	bSlowPull1LifterStn8Down_21 AT %MX30332.21 : BOOL;
	bSlowPull1LifterStn8Down_22 AT %MX30332.22 : BOOL;
	bSlowPull1LifterStn8Down_23 AT %MX30332.23 : BOOL;
	bSlowPull1LifterStn8Down_24 AT %MX30332.24 : BOOL;
	bSlowPull1LifterStn8Down_25 AT %MX30332.25 : BOOL;
	bSlowPull1LifterStn8Down_26 AT %MX30332.26 : BOOL;
	bSlowPull1LifterStn8Down_27 AT %MX30332.27 : BOOL;
	bSlowPull1LifterStn8Down_28 AT %MX30332.28 : BOOL;
	bSlowPull1LifterStn8Down_29 AT %MX30332.29 : BOOL;
	bSlowPull1LifterStn8Down_30 AT %MX30332.30 : BOOL;
	bSlowPull1LifterStn8Down_31 AT %MX30332.31 : BOOL;

	bSlowPull1LifterStn9Down_00 AT %MX30336.0 : BOOL;
	bSlowPull1LifterStn9Down_01 AT %MX30336.1 : BOOL;
	bSlowPull1LifterStn9Down_02 AT %MX30336.2 : BOOL;
	bSlowPull1LifterStn9Down_03 AT %MX30336.3 : BOOL;
	bSlowPull1LifterStn9Down_04 AT %MX30336.4 : BOOL;
	bSlowPull1LifterStn9Down_05 AT %MX30336.5 : BOOL;
	bSlowPull1LifterStn9Down_06 AT %MX30336.6 : BOOL;
	bSlowPull1LifterStn9Down_07 AT %MX30336.7 : BOOL;
	bSlowPull1LifterStn9Down_08 AT %MX30336.8 : BOOL;
	bSlowPull1LifterStn9Down_09 AT %MX30336.9 : BOOL;
	bSlowPull1LifterStn9Down_10 AT %MX30336.10 : BOOL;
	bSlowPull1LifterStn9Down_11 AT %MX30336.11 : BOOL;
	bSlowPull1LifterStn9Down_12 AT %MX30336.12 : BOOL;
	bSlowPull1LifterStn9Down_13 AT %MX30336.13 : BOOL;
	bSlowPull1LifterStn9Down_14 AT %MX30336.14 : BOOL;
	bSlowPull1LifterStn9Down_15 AT %MX30336.15 : BOOL;
	bSlowPull1LifterStn9Down_16 AT %MX30336.16 : BOOL;
	bSlowPull1LifterStn9Down_17 AT %MX30336.17 : BOOL;
	bSlowPull1LifterStn9Down_18 AT %MX30336.18 : BOOL;
	bSlowPull1LifterStn9Down_19 AT %MX30336.19 : BOOL;
	bSlowPull1LifterStn9Down_20 AT %MX30336.20 : BOOL;
	bSlowPull1LifterStn9Down_21 AT %MX30336.21 : BOOL;
	bSlowPull1LifterStn9Down_22 AT %MX30336.22 : BOOL;
	bSlowPull1LifterStn9Down_23 AT %MX30336.23 : BOOL;
	bSlowPull1LifterStn9Down_24 AT %MX30336.24 : BOOL;
	bSlowPull1LifterStn9Down_25 AT %MX30336.25 : BOOL;
	bSlowPull1LifterStn9Down_26 AT %MX30336.26 : BOOL;
	bSlowPull1LifterStn9Down_27 AT %MX30336.27 : BOOL;
	bSlowPull1LifterStn9Down_28 AT %MX30336.28 : BOOL;
	bSlowPull1LifterStn9Down_29 AT %MX30336.29 : BOOL;
	bSlowPull1LifterStn9Down_30 AT %MX30336.30 : BOOL;
	bSlowPull1LifterStn9Down_31 AT %MX30336.31 : BOOL;

	bSlowPull1LifterStn10Down_00 AT %MX30340.0 : BOOL;
	bSlowPull1LifterStn10Down_01 AT %MX30340.1 : BOOL;
	bSlowPull1LifterStn10Down_02 AT %MX30340.2 : BOOL;
	bSlowPull1LifterStn10Down_03 AT %MX30340.3 : BOOL;
	bSlowPull1LifterStn10Down_04 AT %MX30340.4 : BOOL;
	bSlowPull1LifterStn10Down_05 AT %MX30340.5 : BOOL;
	bSlowPull1LifterStn10Down_06 AT %MX30340.6 : BOOL;
	bSlowPull1LifterStn10Down_07 AT %MX30340.7 : BOOL;
	bSlowPull1LifterStn10Down_08 AT %MX30340.8 : BOOL;
	bSlowPull1LifterStn10Down_09 AT %MX30340.9 : BOOL;
	bSlowPull1LifterStn10Down_10 AT %MX30340.10 : BOOL;
	bSlowPull1LifterStn10Down_11 AT %MX30340.11 : BOOL;
	bSlowPull1LifterStn10Down_12 AT %MX30340.12 : BOOL;
	bSlowPull1LifterStn10Down_13 AT %MX30340.13 : BOOL;
	bSlowPull1LifterStn10Down_14 AT %MX30340.14 : BOOL;
	bSlowPull1LifterStn10Down_15 AT %MX30340.15 : BOOL;
	bSlowPull1LifterStn10Down_16 AT %MX30340.16 : BOOL;
	bSlowPull1LifterStn10Down_17 AT %MX30340.17 : BOOL;
	bSlowPull1LifterStn10Down_18 AT %MX30340.18 : BOOL;
	bSlowPull1LifterStn10Down_19 AT %MX30340.19 : BOOL;
	bSlowPull1LifterStn10Down_20 AT %MX30340.20 : BOOL;
	bSlowPull1LifterStn10Down_21 AT %MX30340.21 : BOOL;
	bSlowPull1LifterStn10Down_22 AT %MX30340.22 : BOOL;
	bSlowPull1LifterStn10Down_23 AT %MX30340.23 : BOOL;
	bSlowPull1LifterStn10Down_24 AT %MX30340.24 : BOOL;
	bSlowPull1LifterStn10Down_25 AT %MX30340.25 : BOOL;
	bSlowPull1LifterStn10Down_26 AT %MX30340.26 : BOOL;
	bSlowPull1LifterStn10Down_27 AT %MX30340.27 : BOOL;
	bSlowPull1LifterStn10Down_28 AT %MX30340.28 : BOOL;
	bSlowPull1LifterStn10Down_29 AT %MX30340.29 : BOOL;
	bSlowPull1LifterStn10Down_30 AT %MX30340.30 : BOOL;
	bSlowPull1LifterStn10Down_31 AT %MX30340.31 : BOOL;


(* xxxxxxxxxxxxxxxxxxxxxxxxxxxxxxxxxxxxxxx Lifter xxxxxxxxxxxxxxxxxxxxxxxxxxxxxxxxxxxxxxx*)
(*========= Up/Down LifterAgiUp BOOL LINK with %MX30000-  =========*)

	bSlowPull1LifterStn1AgiUp_00 AT %MX30104.0 : BOOL;
	bSlowPull1LifterStn1AgiUp_01 AT %MX30104.1 : BOOL;
	bSlowPull1LifterStn1AgiUp_02 AT %MX30104.2 : BOOL;
	bSlowPull1LifterStn1AgiUp_03 AT %MX30104.3 : BOOL;
	bSlowPull1LifterStn1AgiUp_04 AT %MX30104.4 : BOOL;
	bSlowPull1LifterStn1AgiUp_05 AT %MX30104.5 : BOOL;
	bSlowPull1LifterStn1AgiUp_06 AT %MX30104.6 : BOOL;
	bSlowPull1LifterStn1AgiUp_07 AT %MX30104.7 : BOOL;
	bSlowPull1LifterStn1AgiUp_08 AT %MX30104.8 : BOOL;
	bSlowPull1LifterStn1AgiUp_09 AT %MX30104.9 : BOOL;
	bSlowPull1LifterStn1AgiUp_10 AT %MX30104.10 : BOOL;
	bSlowPull1LifterStn1AgiUp_11 AT %MX30104.11 : BOOL;
	bSlowPull1LifterStn1AgiUp_12 AT %MX30104.12 : BOOL;
	bSlowPull1LifterStn1AgiUp_13 AT %MX30104.13 : BOOL;
	bSlowPull1LifterStn1AgiUp_14 AT %MX30104.14 : BOOL;
	bSlowPull1LifterStn1AgiUp_15 AT %MX30104.15 : BOOL;
	bSlowPull1LifterStn1AgiUp_16 AT %MX30104.16 : BOOL;
	bSlowPull1LifterStn1AgiUp_17 AT %MX30104.17 : BOOL;
	bSlowPull1LifterStn1AgiUp_18 AT %MX30104.18 : BOOL;
	bSlowPull1LifterStn1AgiUp_19 AT %MX30104.19 : BOOL;
	bSlowPull1LifterStn1AgiUp_20 AT %MX30104.20 : BOOL;
	bSlowPull1LifterStn1AgiUp_21 AT %MX30104.21 : BOOL;
	bSlowPull1LifterStn1AgiUp_22 AT %MX30104.22 : BOOL;
	bSlowPull1LifterStn1AgiUp_23 AT %MX30104.23 : BOOL;
	bSlowPull1LifterStn1AgiUp_24 AT %MX30104.24 : BOOL;
	bSlowPull1LifterStn1AgiUp_25 AT %MX30104.25 : BOOL;
	bSlowPull1LifterStn1AgiUp_26 AT %MX30104.26 : BOOL;
	bSlowPull1LifterStn1AgiUp_27 AT %MX30104.27 : BOOL;
	bSlowPull1LifterStn1AgiUp_28 AT %MX30104.28 : BOOL;
	bSlowPull1LifterStn1AgiUp_29 AT %MX30104.29 : BOOL;
	bSlowPull1LifterStn1AgiUp_30 AT %MX30104.30 : BOOL;
	bSlowPull1LifterStn1AgiUp_31 AT %MX30104.31 : BOOL;

	bSlowPull1LifterStn2AgiUp_00 AT %MX30108.0 : BOOL;
	bSlowPull1LifterStn2AgiUp_01 AT %MX30108.1 : BOOL;
	bSlowPull1LifterStn2AgiUp_02 AT %MX30108.2 : BOOL;
	bSlowPull1LifterStn2AgiUp_03 AT %MX30108.3 : BOOL;
	bSlowPull1LifterStn2AgiUp_04 AT %MX30108.4 : BOOL;
	bSlowPull1LifterStn2AgiUp_05 AT %MX30108.5 : BOOL;
	bSlowPull1LifterStn2AgiUp_06 AT %MX30108.6 : BOOL;
	bSlowPull1LifterStn2AgiUp_07 AT %MX30108.7 : BOOL;
	bSlowPull1LifterStn2AgiUp_08 AT %MX30108.8 : BOOL;
	bSlowPull1LifterStn2AgiUp_09 AT %MX30108.9 : BOOL;
	bSlowPull1LifterStn2AgiUp_10 AT %MX30108.10 : BOOL;
	bSlowPull1LifterStn2AgiUp_11 AT %MX30108.11 : BOOL;
	bSlowPull1LifterStn2AgiUp_12 AT %MX30108.12 : BOOL;
	bSlowPull1LifterStn2AgiUp_13 AT %MX30108.13 : BOOL;
	bSlowPull1LifterStn2AgiUp_14 AT %MX30108.14 : BOOL;
	bSlowPull1LifterStn2AgiUp_15 AT %MX30108.15 : BOOL;
	bSlowPull1LifterStn2AgiUp_16 AT %MX30108.16 : BOOL;
	bSlowPull1LifterStn2AgiUp_17 AT %MX30108.17 : BOOL;
	bSlowPull1LifterStn2AgiUp_18 AT %MX30108.18 : BOOL;
	bSlowPull1LifterStn2AgiUp_19 AT %MX30108.19 : BOOL;
	bSlowPull1LifterStn2AgiUp_20 AT %MX30108.20 : BOOL;
	bSlowPull1LifterStn2AgiUp_21 AT %MX30108.21 : BOOL;
	bSlowPull1LifterStn2AgiUp_22 AT %MX30108.22 : BOOL;
	bSlowPull1LifterStn2AgiUp_23 AT %MX30108.23 : BOOL;
	bSlowPull1LifterStn2AgiUp_24 AT %MX30108.24 : BOOL;
	bSlowPull1LifterStn2AgiUp_25 AT %MX30108.25 : BOOL;
	bSlowPull1LifterStn2AgiUp_26 AT %MX30108.26 : BOOL;
	bSlowPull1LifterStn2AgiUp_27 AT %MX30108.27 : BOOL;
	bSlowPull1LifterStn2AgiUp_28 AT %MX30108.28 : BOOL;
	bSlowPull1LifterStn2AgiUp_29 AT %MX30108.29 : BOOL;
	bSlowPull1LifterStn2AgiUp_30 AT %MX30108.30 : BOOL;
	bSlowPull1LifterStn2AgiUp_31 AT %MX30108.31 : BOOL;

	bSlowPull1LifterStn3AgiUp_00 AT %MX30112.0 : BOOL;
	bSlowPull1LifterStn3AgiUp_01 AT %MX30112.1 : BOOL;
	bSlowPull1LifterStn3AgiUp_02 AT %MX30112.2 : BOOL;
	bSlowPull1LifterStn3AgiUp_03 AT %MX30112.3 : BOOL;
	bSlowPull1LifterStn3AgiUp_04 AT %MX30112.4 : BOOL;
	bSlowPull1LifterStn3AgiUp_05 AT %MX30112.5 : BOOL;
	bSlowPull1LifterStn3AgiUp_06 AT %MX30112.6 : BOOL;
	bSlowPull1LifterStn3AgiUp_07 AT %MX30112.7 : BOOL;
	bSlowPull1LifterStn3AgiUp_08 AT %MX30112.8 : BOOL;
	bSlowPull1LifterStn3AgiUp_09 AT %MX30112.9 : BOOL;
	bSlowPull1LifterStn3AgiUp_10 AT %MX30112.10 : BOOL;
	bSlowPull1LifterStn3AgiUp_11 AT %MX30112.11 : BOOL;
	bSlowPull1LifterStn3AgiUp_12 AT %MX30112.12 : BOOL;
	bSlowPull1LifterStn3AgiUp_13 AT %MX30112.13 : BOOL;
	bSlowPull1LifterStn3AgiUp_14 AT %MX30112.14 : BOOL;
	bSlowPull1LifterStn3AgiUp_15 AT %MX30112.15 : BOOL;
	bSlowPull1LifterStn3AgiUp_16 AT %MX30112.16 : BOOL;
	bSlowPull1LifterStn3AgiUp_17 AT %MX30112.17 : BOOL;
	bSlowPull1LifterStn3AgiUp_18 AT %MX30112.18 : BOOL;
	bSlowPull1LifterStn3AgiUp_19 AT %MX30112.19 : BOOL;
	bSlowPull1LifterStn3AgiUp_20 AT %MX30112.20 : BOOL;
	bSlowPull1LifterStn3AgiUp_21 AT %MX30112.21 : BOOL;
	bSlowPull1LifterStn3AgiUp_22 AT %MX30112.22 : BOOL;
	bSlowPull1LifterStn3AgiUp_23 AT %MX30112.23 : BOOL;
	bSlowPull1LifterStn3AgiUp_24 AT %MX30112.24 : BOOL;
	bSlowPull1LifterStn3AgiUp_25 AT %MX30112.25 : BOOL;
	bSlowPull1LifterStn3AgiUp_26 AT %MX30112.26 : BOOL;
	bSlowPull1LifterStn3AgiUp_27 AT %MX30112.27 : BOOL;
	bSlowPull1LifterStn3AgiUp_28 AT %MX30112.28 : BOOL;
	bSlowPull1LifterStn3AgiUp_29 AT %MX30112.29 : BOOL;
	bSlowPull1LifterStn3AgiUp_30 AT %MX30112.30 : BOOL;
	bSlowPull1LifterStn3AgiUp_31 AT %MX30112.31 : BOOL;

	bSlowPull1LifterStn4AgiUp_00 AT %MX30116.0 : BOOL;
	bSlowPull1LifterStn4AgiUp_01 AT %MX30116.1 : BOOL;
	bSlowPull1LifterStn4AgiUp_02 AT %MX30116.2 : BOOL;
	bSlowPull1LifterStn4AgiUp_03 AT %MX30116.3 : BOOL;
	bSlowPull1LifterStn4AgiUp_04 AT %MX30116.4 : BOOL;
	bSlowPull1LifterStn4AgiUp_05 AT %MX30116.5 : BOOL;
	bSlowPull1LifterStn4AgiUp_06 AT %MX30116.6 : BOOL;
	bSlowPull1LifterStn4AgiUp_07 AT %MX30116.7 : BOOL;
	bSlowPull1LifterStn4AgiUp_08 AT %MX30116.8 : BOOL;
	bSlowPull1LifterStn4AgiUp_09 AT %MX30116.9 : BOOL;
	bSlowPull1LifterStn4AgiUp_10 AT %MX30116.10 : BOOL;
	bSlowPull1LifterStn4AgiUp_11 AT %MX30116.11 : BOOL;
	bSlowPull1LifterStn4AgiUp_12 AT %MX30116.12 : BOOL;
	bSlowPull1LifterStn4AgiUp_13 AT %MX30116.13 : BOOL;
	bSlowPull1LifterStn4AgiUp_14 AT %MX30116.14 : BOOL;
	bSlowPull1LifterStn4AgiUp_15 AT %MX30116.15 : BOOL;
	bSlowPull1LifterStn4AgiUp_16 AT %MX30116.16 : BOOL;
	bSlowPull1LifterStn4AgiUp_17 AT %MX30116.17 : BOOL;
	bSlowPull1LifterStn4AgiUp_18 AT %MX30116.18 : BOOL;
	bSlowPull1LifterStn4AgiUp_19 AT %MX30116.19 : BOOL;
	bSlowPull1LifterStn4AgiUp_20 AT %MX30116.20 : BOOL;
	bSlowPull1LifterStn4AgiUp_21 AT %MX30116.21 : BOOL;
	bSlowPull1LifterStn4AgiUp_22 AT %MX30116.22 : BOOL;
	bSlowPull1LifterStn4AgiUp_23 AT %MX30116.23 : BOOL;
	bSlowPull1LifterStn4AgiUp_24 AT %MX30116.24 : BOOL;
	bSlowPull1LifterStn4AgiUp_25 AT %MX30116.25 : BOOL;
	bSlowPull1LifterStn4AgiUp_26 AT %MX30116.26 : BOOL;
	bSlowPull1LifterStn4AgiUp_27 AT %MX30116.27 : BOOL;
	bSlowPull1LifterStn4AgiUp_28 AT %MX30116.28 : BOOL;
	bSlowPull1LifterStn4AgiUp_29 AT %MX30116.29 : BOOL;
	bSlowPull1LifterStn4AgiUp_30 AT %MX30116.30 : BOOL;
	bSlowPull1LifterStn4AgiUp_31 AT %MX30116.31 : BOOL;

	bSlowPull1LifterStn5AgiUp_00 AT %MX30120.0 : BOOL;
	bSlowPull1LifterStn5AgiUp_01 AT %MX30120.1 : BOOL;
	bSlowPull1LifterStn5AgiUp_02 AT %MX30120.2 : BOOL;
	bSlowPull1LifterStn5AgiUp_03 AT %MX30120.3 : BOOL;
	bSlowPull1LifterStn5AgiUp_04 AT %MX30120.4 : BOOL;
	bSlowPull1LifterStn5AgiUp_05 AT %MX30120.5 : BOOL;
	bSlowPull1LifterStn5AgiUp_06 AT %MX30120.6 : BOOL;
	bSlowPull1LifterStn5AgiUp_07 AT %MX30120.7 : BOOL;
	bSlowPull1LifterStn5AgiUp_08 AT %MX30120.8 : BOOL;
	bSlowPull1LifterStn5AgiUp_09 AT %MX30120.9 : BOOL;
	bSlowPull1LifterStn5AgiUp_10 AT %MX30120.10 : BOOL;
	bSlowPull1LifterStn5AgiUp_11 AT %MX30120.11 : BOOL;
	bSlowPull1LifterStn5AgiUp_12 AT %MX30120.12 : BOOL;
	bSlowPull1LifterStn5AgiUp_13 AT %MX30120.13 : BOOL;
	bSlowPull1LifterStn5AgiUp_14 AT %MX30120.14 : BOOL;
	bSlowPull1LifterStn5AgiUp_15 AT %MX30120.15 : BOOL;
	bSlowPull1LifterStn5AgiUp_16 AT %MX30120.16 : BOOL;
	bSlowPull1LifterStn5AgiUp_17 AT %MX30120.17 : BOOL;
	bSlowPull1LifterStn5AgiUp_18 AT %MX30120.18 : BOOL;
	bSlowPull1LifterStn5AgiUp_19 AT %MX30120.19 : BOOL;
	bSlowPull1LifterStn5AgiUp_20 AT %MX30120.20 : BOOL;
	bSlowPull1LifterStn5AgiUp_21 AT %MX30120.21 : BOOL;
	bSlowPull1LifterStn5AgiUp_22 AT %MX30120.22 : BOOL;
	bSlowPull1LifterStn5AgiUp_23 AT %MX30120.23 : BOOL;
	bSlowPull1LifterStn5AgiUp_24 AT %MX30120.24 : BOOL;
	bSlowPull1LifterStn5AgiUp_25 AT %MX30120.25 : BOOL;
	bSlowPull1LifterStn5AgiUp_26 AT %MX30120.26 : BOOL;
	bSlowPull1LifterStn5AgiUp_27 AT %MX30120.27 : BOOL;
	bSlowPull1LifterStn5AgiUp_28 AT %MX30120.28 : BOOL;
	bSlowPull1LifterStn5AgiUp_29 AT %MX30120.29 : BOOL;
	bSlowPull1LifterStn5AgiUp_30 AT %MX30120.30 : BOOL;
	bSlowPull1LifterStn5AgiUp_31 AT %MX30120.31 : BOOL;

	bSlowPull1LifterStn6AgiUp_00 AT %MX30124.0 : BOOL;
	bSlowPull1LifterStn6AgiUp_01 AT %MX30124.1 : BOOL;
	bSlowPull1LifterStn6AgiUp_02 AT %MX30124.2 : BOOL;
	bSlowPull1LifterStn6AgiUp_03 AT %MX30124.3 : BOOL;
	bSlowPull1LifterStn6AgiUp_04 AT %MX30124.4 : BOOL;
	bSlowPull1LifterStn6AgiUp_05 AT %MX30124.5 : BOOL;
	bSlowPull1LifterStn6AgiUp_06 AT %MX30124.6 : BOOL;
	bSlowPull1LifterStn6AgiUp_07 AT %MX30124.7 : BOOL;
	bSlowPull1LifterStn6AgiUp_08 AT %MX30124.8 : BOOL;
	bSlowPull1LifterStn6AgiUp_09 AT %MX30124.9 : BOOL;
	bSlowPull1LifterStn6AgiUp_10 AT %MX30124.10 : BOOL;
	bSlowPull1LifterStn6AgiUp_11 AT %MX30124.11 : BOOL;
	bSlowPull1LifterStn6AgiUp_12 AT %MX30124.12 : BOOL;
	bSlowPull1LifterStn6AgiUp_13 AT %MX30124.13 : BOOL;
	bSlowPull1LifterStn6AgiUp_14 AT %MX30124.14 : BOOL;
	bSlowPull1LifterStn6AgiUp_15 AT %MX30124.15 : BOOL;
	bSlowPull1LifterStn6AgiUp_16 AT %MX30124.16 : BOOL;
	bSlowPull1LifterStn6AgiUp_17 AT %MX30124.17 : BOOL;
	bSlowPull1LifterStn6AgiUp_18 AT %MX30124.18 : BOOL;
	bSlowPull1LifterStn6AgiUp_19 AT %MX30124.19 : BOOL;
	bSlowPull1LifterStn6AgiUp_20 AT %MX30124.20 : BOOL;
	bSlowPull1LifterStn6AgiUp_21 AT %MX30124.21 : BOOL;
	bSlowPull1LifterStn6AgiUp_22 AT %MX30124.22 : BOOL;
	bSlowPull1LifterStn6AgiUp_23 AT %MX30124.23 : BOOL;
	bSlowPull1LifterStn6AgiUp_24 AT %MX30124.24 : BOOL;
	bSlowPull1LifterStn6AgiUp_25 AT %MX30124.25 : BOOL;
	bSlowPull1LifterStn6AgiUp_26 AT %MX30124.26 : BOOL;
	bSlowPull1LifterStn6AgiUp_27 AT %MX30124.27 : BOOL;
	bSlowPull1LifterStn6AgiUp_28 AT %MX30124.28 : BOOL;
	bSlowPull1LifterStn6AgiUp_29 AT %MX30124.29 : BOOL;
	bSlowPull1LifterStn6AgiUp_30 AT %MX30124.30 : BOOL;
	bSlowPull1LifterStn6AgiUp_31 AT %MX30124.31 : BOOL;

	bSlowPull1LifterStn7AgiUp_00 AT %MX30128.0 : BOOL;
	bSlowPull1LifterStn7AgiUp_01 AT %MX30128.1 : BOOL;
	bSlowPull1LifterStn7AgiUp_02 AT %MX30128.2 : BOOL;
	bSlowPull1LifterStn7AgiUp_03 AT %MX30128.3 : BOOL;
	bSlowPull1LifterStn7AgiUp_04 AT %MX30128.4 : BOOL;
	bSlowPull1LifterStn7AgiUp_05 AT %MX30128.5 : BOOL;
	bSlowPull1LifterStn7AgiUp_06 AT %MX30128.6 : BOOL;
	bSlowPull1LifterStn7AgiUp_07 AT %MX30128.7 : BOOL;
	bSlowPull1LifterStn7AgiUp_08 AT %MX30128.8 : BOOL;
	bSlowPull1LifterStn7AgiUp_09 AT %MX30128.9 : BOOL;
	bSlowPull1LifterStn7AgiUp_10 AT %MX30128.10 : BOOL;
	bSlowPull1LifterStn7AgiUp_11 AT %MX30128.11 : BOOL;
	bSlowPull1LifterStn7AgiUp_12 AT %MX30128.12 : BOOL;
	bSlowPull1LifterStn7AgiUp_13 AT %MX30128.13 : BOOL;
	bSlowPull1LifterStn7AgiUp_14 AT %MX30128.14 : BOOL;
	bSlowPull1LifterStn7AgiUp_15 AT %MX30128.15 : BOOL;
	bSlowPull1LifterStn7AgiUp_16 AT %MX30128.16 : BOOL;
	bSlowPull1LifterStn7AgiUp_17 AT %MX30128.17 : BOOL;
	bSlowPull1LifterStn7AgiUp_18 AT %MX30128.18 : BOOL;
	bSlowPull1LifterStn7AgiUp_19 AT %MX30128.19 : BOOL;
	bSlowPull1LifterStn7AgiUp_20 AT %MX30128.20 : BOOL;
	bSlowPull1LifterStn7AgiUp_21 AT %MX30128.21 : BOOL;
	bSlowPull1LifterStn7AgiUp_22 AT %MX30128.22 : BOOL;
	bSlowPull1LifterStn7AgiUp_23 AT %MX30128.23 : BOOL;
	bSlowPull1LifterStn7AgiUp_24 AT %MX30128.24 : BOOL;
	bSlowPull1LifterStn7AgiUp_25 AT %MX30128.25 : BOOL;
	bSlowPull1LifterStn7AgiUp_26 AT %MX30128.26 : BOOL;
	bSlowPull1LifterStn7AgiUp_27 AT %MX30128.27 : BOOL;
	bSlowPull1LifterStn7AgiUp_28 AT %MX30128.28 : BOOL;
	bSlowPull1LifterStn7AgiUp_29 AT %MX30128.29 : BOOL;
	bSlowPull1LifterStn7AgiUp_30 AT %MX30128.30 : BOOL;
	bSlowPull1LifterStn7AgiUp_31 AT %MX30128.31 : BOOL;

	bSlowPull1LifterStn8AgiUp_00 AT %MX30132.0 : BOOL;
	bSlowPull1LifterStn8AgiUp_01 AT %MX30132.1 : BOOL;
	bSlowPull1LifterStn8AgiUp_02 AT %MX30132.2 : BOOL;
	bSlowPull1LifterStn8AgiUp_03 AT %MX30132.3 : BOOL;
	bSlowPull1LifterStn8AgiUp_04 AT %MX30132.4 : BOOL;
	bSlowPull1LifterStn8AgiUp_05 AT %MX30132.5 : BOOL;
	bSlowPull1LifterStn8AgiUp_06 AT %MX30132.6 : BOOL;
	bSlowPull1LifterStn8AgiUp_07 AT %MX30132.7 : BOOL;
	bSlowPull1LifterStn8AgiUp_08 AT %MX30132.8 : BOOL;
	bSlowPull1LifterStn8AgiUp_09 AT %MX30132.9 : BOOL;
	bSlowPull1LifterStn8AgiUp_10 AT %MX30132.10 : BOOL;
	bSlowPull1LifterStn8AgiUp_11 AT %MX30132.11 : BOOL;
	bSlowPull1LifterStn8AgiUp_12 AT %MX30132.12 : BOOL;
	bSlowPull1LifterStn8AgiUp_13 AT %MX30132.13 : BOOL;
	bSlowPull1LifterStn8AgiUp_14 AT %MX30132.14 : BOOL;
	bSlowPull1LifterStn8AgiUp_15 AT %MX30132.15 : BOOL;
	bSlowPull1LifterStn8AgiUp_16 AT %MX30132.16 : BOOL;
	bSlowPull1LifterStn8AgiUp_17 AT %MX30132.17 : BOOL;
	bSlowPull1LifterStn8AgiUp_18 AT %MX30132.18 : BOOL;
	bSlowPull1LifterStn8AgiUp_19 AT %MX30132.19 : BOOL;
	bSlowPull1LifterStn8AgiUp_20 AT %MX30132.20 : BOOL;
	bSlowPull1LifterStn8AgiUp_21 AT %MX30132.21 : BOOL;
	bSlowPull1LifterStn8AgiUp_22 AT %MX30132.22 : BOOL;
	bSlowPull1LifterStn8AgiUp_23 AT %MX30132.23 : BOOL;
	bSlowPull1LifterStn8AgiUp_24 AT %MX30132.24 : BOOL;
	bSlowPull1LifterStn8AgiUp_25 AT %MX30132.25 : BOOL;
	bSlowPull1LifterStn8AgiUp_26 AT %MX30132.26 : BOOL;
	bSlowPull1LifterStn8AgiUp_27 AT %MX30132.27 : BOOL;
	bSlowPull1LifterStn8AgiUp_28 AT %MX30132.28 : BOOL;
	bSlowPull1LifterStn8AgiUp_29 AT %MX30132.29 : BOOL;
	bSlowPull1LifterStn8AgiUp_30 AT %MX30132.30 : BOOL;
	bSlowPull1LifterStn8AgiUp_31 AT %MX30132.31 : BOOL;

	bSlowPull1LifterStn9AgiUp_00 AT %MX30136.0 : BOOL;
	bSlowPull1LifterStn9AgiUp_01 AT %MX30136.1 : BOOL;
	bSlowPull1LifterStn9AgiUp_02 AT %MX30136.2 : BOOL;
	bSlowPull1LifterStn9AgiUp_03 AT %MX30136.3 : BOOL;
	bSlowPull1LifterStn9AgiUp_04 AT %MX30136.4 : BOOL;
	bSlowPull1LifterStn9AgiUp_05 AT %MX30136.5 : BOOL;
	bSlowPull1LifterStn9AgiUp_06 AT %MX30136.6 : BOOL;
	bSlowPull1LifterStn9AgiUp_07 AT %MX30136.7 : BOOL;
	bSlowPull1LifterStn9AgiUp_08 AT %MX30136.8 : BOOL;
	bSlowPull1LifterStn9AgiUp_09 AT %MX30136.9 : BOOL;
	bSlowPull1LifterStn9AgiUp_10 AT %MX30136.10 : BOOL;
	bSlowPull1LifterStn9AgiUp_11 AT %MX30136.11 : BOOL;
	bSlowPull1LifterStn9AgiUp_12 AT %MX30136.12 : BOOL;
	bSlowPull1LifterStn9AgiUp_13 AT %MX30136.13 : BOOL;
	bSlowPull1LifterStn9AgiUp_14 AT %MX30136.14 : BOOL;
	bSlowPull1LifterStn9AgiUp_15 AT %MX30136.15 : BOOL;
	bSlowPull1LifterStn9AgiUp_16 AT %MX30136.16 : BOOL;
	bSlowPull1LifterStn9AgiUp_17 AT %MX30136.17 : BOOL;
	bSlowPull1LifterStn9AgiUp_18 AT %MX30136.18 : BOOL;
	bSlowPull1LifterStn9AgiUp_19 AT %MX30136.19 : BOOL;
	bSlowPull1LifterStn9AgiUp_20 AT %MX30136.20 : BOOL;
	bSlowPull1LifterStn9AgiUp_21 AT %MX30136.21 : BOOL;
	bSlowPull1LifterStn9AgiUp_22 AT %MX30136.22 : BOOL;
	bSlowPull1LifterStn9AgiUp_23 AT %MX30136.23 : BOOL;
	bSlowPull1LifterStn9AgiUp_24 AT %MX30136.24 : BOOL;
	bSlowPull1LifterStn9AgiUp_25 AT %MX30136.25 : BOOL;
	bSlowPull1LifterStn9AgiUp_26 AT %MX30136.26 : BOOL;
	bSlowPull1LifterStn9AgiUp_27 AT %MX30136.27 : BOOL;
	bSlowPull1LifterStn9AgiUp_28 AT %MX30136.28 : BOOL;
	bSlowPull1LifterStn9AgiUp_29 AT %MX30136.29 : BOOL;
	bSlowPull1LifterStn9AgiUp_30 AT %MX30136.30 : BOOL;
	bSlowPull1LifterStn9AgiUp_31 AT %MX30136.31 : BOOL;

	bSlowPull1LifterStn10AgiUp_00 AT %MX30140.0 : BOOL;
	bSlowPull1LifterStn10AgiUp_01 AT %MX30140.1 : BOOL;
	bSlowPull1LifterStn10AgiUp_02 AT %MX30140.2 : BOOL;
	bSlowPull1LifterStn10AgiUp_03 AT %MX30140.3 : BOOL;
	bSlowPull1LifterStn10AgiUp_04 AT %MX30140.4 : BOOL;
	bSlowPull1LifterStn10AgiUp_05 AT %MX30140.5 : BOOL;
	bSlowPull1LifterStn10AgiUp_06 AT %MX30140.6 : BOOL;
	bSlowPull1LifterStn10AgiUp_07 AT %MX30140.7 : BOOL;
	bSlowPull1LifterStn10AgiUp_08 AT %MX30140.8 : BOOL;
	bSlowPull1LifterStn10AgiUp_09 AT %MX30140.9 : BOOL;
	bSlowPull1LifterStn10AgiUp_10 AT %MX30140.10 : BOOL;
	bSlowPull1LifterStn10AgiUp_11 AT %MX30140.11 : BOOL;
	bSlowPull1LifterStn10AgiUp_12 AT %MX30140.12 : BOOL;
	bSlowPull1LifterStn10AgiUp_13 AT %MX30140.13 : BOOL;
	bSlowPull1LifterStn10AgiUp_14 AT %MX30140.14 : BOOL;
	bSlowPull1LifterStn10AgiUp_15 AT %MX30140.15 : BOOL;
	bSlowPull1LifterStn10AgiUp_16 AT %MX30140.16 : BOOL;
	bSlowPull1LifterStn10AgiUp_17 AT %MX30140.17 : BOOL;
	bSlowPull1LifterStn10AgiUp_18 AT %MX30140.18 : BOOL;
	bSlowPull1LifterStn10AgiUp_19 AT %MX30140.19 : BOOL;
	bSlowPull1LifterStn10AgiUp_20 AT %MX30140.20 : BOOL;
	bSlowPull1LifterStn10AgiUp_21 AT %MX30140.21 : BOOL;
	bSlowPull1LifterStn10AgiUp_22 AT %MX30140.22 : BOOL;
	bSlowPull1LifterStn10AgiUp_23 AT %MX30140.23 : BOOL;
	bSlowPull1LifterStn10AgiUp_24 AT %MX30140.24 : BOOL;
	bSlowPull1LifterStn10AgiUp_25 AT %MX30140.25 : BOOL;
	bSlowPull1LifterStn10AgiUp_26 AT %MX30140.26 : BOOL;
	bSlowPull1LifterStn10AgiUp_27 AT %MX30140.27 : BOOL;
	bSlowPull1LifterStn10AgiUp_28 AT %MX30140.28 : BOOL;
	bSlowPull1LifterStn10AgiUp_29 AT %MX30140.29 : BOOL;
	bSlowPull1LifterStn10AgiUp_30 AT %MX30140.30 : BOOL;
	bSlowPull1LifterStn10AgiUp_31 AT %MX30140.31 : BOOL;


(* xxxxxxxxxxxxxxxxxxxxxxxxxxxxxxxxxxxxxxx Lifter xxxxxxxxxxxxxxxxxxxxxxxxxxxxxxxxxxxxxxx*)
(*========= Up/Down LifterAgiDown BOOL LINK with %MX30000-  =========*)

	bSlowPull1LifterStn1AgiDown_00 AT %MX30204.0 : BOOL;
	bSlowPull1LifterStn1AgiDown_01 AT %MX30204.1 : BOOL;
	bSlowPull1LifterStn1AgiDown_02 AT %MX30204.2 : BOOL;
	bSlowPull1LifterStn1AgiDown_03 AT %MX30204.3 : BOOL;
	bSlowPull1LifterStn1AgiDown_04 AT %MX30204.4 : BOOL;
	bSlowPull1LifterStn1AgiDown_05 AT %MX30204.5 : BOOL;
	bSlowPull1LifterStn1AgiDown_06 AT %MX30204.6 : BOOL;
	bSlowPull1LifterStn1AgiDown_07 AT %MX30204.7 : BOOL;
	bSlowPull1LifterStn1AgiDown_08 AT %MX30204.8 : BOOL;
	bSlowPull1LifterStn1AgiDown_09 AT %MX30204.9 : BOOL;
	bSlowPull1LifterStn1AgiDown_10 AT %MX30204.10 : BOOL;
	bSlowPull1LifterStn1AgiDown_11 AT %MX30204.11 : BOOL;
	bSlowPull1LifterStn1AgiDown_12 AT %MX30204.12 : BOOL;
	bSlowPull1LifterStn1AgiDown_13 AT %MX30204.13 : BOOL;
	bSlowPull1LifterStn1AgiDown_14 AT %MX30204.14 : BOOL;
	bSlowPull1LifterStn1AgiDown_15 AT %MX30204.15 : BOOL;
	bSlowPull1LifterStn1AgiDown_16 AT %MX30204.16 : BOOL;
	bSlowPull1LifterStn1AgiDown_17 AT %MX30204.17 : BOOL;
	bSlowPull1LifterStn1AgiDown_18 AT %MX30204.18 : BOOL;
	bSlowPull1LifterStn1AgiDown_19 AT %MX30204.19 : BOOL;
	bSlowPull1LifterStn1AgiDown_20 AT %MX30204.20 : BOOL;
	bSlowPull1LifterStn1AgiDown_21 AT %MX30204.21 : BOOL;
	bSlowPull1LifterStn1AgiDown_22 AT %MX30204.22 : BOOL;
	bSlowPull1LifterStn1AgiDown_23 AT %MX30204.23 : BOOL;
	bSlowPull1LifterStn1AgiDown_24 AT %MX30204.24 : BOOL;
	bSlowPull1LifterStn1AgiDown_25 AT %MX30204.25 : BOOL;
	bSlowPull1LifterStn1AgiDown_26 AT %MX30204.26 : BOOL;
	bSlowPull1LifterStn1AgiDown_27 AT %MX30204.27 : BOOL;
	bSlowPull1LifterStn1AgiDown_28 AT %MX30204.28 : BOOL;
	bSlowPull1LifterStn1AgiDown_29 AT %MX30204.29 : BOOL;
	bSlowPull1LifterStn1AgiDown_30 AT %MX30204.30 : BOOL;
	bSlowPull1LifterStn1AgiDown_31 AT %MX30204.31 : BOOL;

	bSlowPull1LifterStn2AgiDown_00 AT %MX30208.0 : BOOL;
	bSlowPull1LifterStn2AgiDown_01 AT %MX30208.1 : BOOL;
	bSlowPull1LifterStn2AgiDown_02 AT %MX30208.2 : BOOL;
	bSlowPull1LifterStn2AgiDown_03 AT %MX30208.3 : BOOL;
	bSlowPull1LifterStn2AgiDown_04 AT %MX30208.4 : BOOL;
	bSlowPull1LifterStn2AgiDown_05 AT %MX30208.5 : BOOL;
	bSlowPull1LifterStn2AgiDown_06 AT %MX30208.6 : BOOL;
	bSlowPull1LifterStn2AgiDown_07 AT %MX30208.7 : BOOL;
	bSlowPull1LifterStn2AgiDown_08 AT %MX30208.8 : BOOL;
	bSlowPull1LifterStn2AgiDown_09 AT %MX30208.9 : BOOL;
	bSlowPull1LifterStn2AgiDown_10 AT %MX30208.10 : BOOL;
	bSlowPull1LifterStn2AgiDown_11 AT %MX30208.11 : BOOL;
	bSlowPull1LifterStn2AgiDown_12 AT %MX30208.12 : BOOL;
	bSlowPull1LifterStn2AgiDown_13 AT %MX30208.13 : BOOL;
	bSlowPull1LifterStn2AgiDown_14 AT %MX30208.14 : BOOL;
	bSlowPull1LifterStn2AgiDown_15 AT %MX30208.15 : BOOL;
	bSlowPull1LifterStn2AgiDown_16 AT %MX30208.16 : BOOL;
	bSlowPull1LifterStn2AgiDown_17 AT %MX30208.17 : BOOL;
	bSlowPull1LifterStn2AgiDown_18 AT %MX30208.18 : BOOL;
	bSlowPull1LifterStn2AgiDown_19 AT %MX30208.19 : BOOL;
	bSlowPull1LifterStn2AgiDown_20 AT %MX30208.20 : BOOL;
	bSlowPull1LifterStn2AgiDown_21 AT %MX30208.21 : BOOL;
	bSlowPull1LifterStn2AgiDown_22 AT %MX30208.22 : BOOL;
	bSlowPull1LifterStn2AgiDown_23 AT %MX30208.23 : BOOL;
	bSlowPull1LifterStn2AgiDown_24 AT %MX30208.24 : BOOL;
	bSlowPull1LifterStn2AgiDown_25 AT %MX30208.25 : BOOL;
	bSlowPull1LifterStn2AgiDown_26 AT %MX30208.26 : BOOL;
	bSlowPull1LifterStn2AgiDown_27 AT %MX30208.27 : BOOL;
	bSlowPull1LifterStn2AgiDown_28 AT %MX30208.28 : BOOL;
	bSlowPull1LifterStn2AgiDown_29 AT %MX30208.29 : BOOL;
	bSlowPull1LifterStn2AgiDown_30 AT %MX30208.30 : BOOL;
	bSlowPull1LifterStn2AgiDown_31 AT %MX30208.31 : BOOL;

	bSlowPull1LifterStn3AgiDown_00 AT %MX30212.0 : BOOL;
	bSlowPull1LifterStn3AgiDown_01 AT %MX30212.1 : BOOL;
	bSlowPull1LifterStn3AgiDown_02 AT %MX30212.2 : BOOL;
	bSlowPull1LifterStn3AgiDown_03 AT %MX30212.3 : BOOL;
	bSlowPull1LifterStn3AgiDown_04 AT %MX30212.4 : BOOL;
	bSlowPull1LifterStn3AgiDown_05 AT %MX30212.5 : BOOL;
	bSlowPull1LifterStn3AgiDown_06 AT %MX30212.6 : BOOL;
	bSlowPull1LifterStn3AgiDown_07 AT %MX30212.7 : BOOL;
	bSlowPull1LifterStn3AgiDown_08 AT %MX30212.8 : BOOL;
	bSlowPull1LifterStn3AgiDown_09 AT %MX30212.9 : BOOL;
	bSlowPull1LifterStn3AgiDown_10 AT %MX30212.10 : BOOL;
	bSlowPull1LifterStn3AgiDown_11 AT %MX30212.11 : BOOL;
	bSlowPull1LifterStn3AgiDown_12 AT %MX30212.12 : BOOL;
	bSlowPull1LifterStn3AgiDown_13 AT %MX30212.13 : BOOL;
	bSlowPull1LifterStn3AgiDown_14 AT %MX30212.14 : BOOL;
	bSlowPull1LifterStn3AgiDown_15 AT %MX30212.15 : BOOL;
	bSlowPull1LifterStn3AgiDown_16 AT %MX30212.16 : BOOL;
	bSlowPull1LifterStn3AgiDown_17 AT %MX30212.17 : BOOL;
	bSlowPull1LifterStn3AgiDown_18 AT %MX30212.18 : BOOL;
	bSlowPull1LifterStn3AgiDown_19 AT %MX30212.19 : BOOL;
	bSlowPull1LifterStn3AgiDown_20 AT %MX30212.20 : BOOL;
	bSlowPull1LifterStn3AgiDown_21 AT %MX30212.21 : BOOL;
	bSlowPull1LifterStn3AgiDown_22 AT %MX30212.22 : BOOL;
	bSlowPull1LifterStn3AgiDown_23 AT %MX30212.23 : BOOL;
	bSlowPull1LifterStn3AgiDown_24 AT %MX30212.24 : BOOL;
	bSlowPull1LifterStn3AgiDown_25 AT %MX30212.25 : BOOL;
	bSlowPull1LifterStn3AgiDown_26 AT %MX30212.26 : BOOL;
	bSlowPull1LifterStn3AgiDown_27 AT %MX30212.27 : BOOL;
	bSlowPull1LifterStn3AgiDown_28 AT %MX30212.28 : BOOL;
	bSlowPull1LifterStn3AgiDown_29 AT %MX30212.29 : BOOL;
	bSlowPull1LifterStn3AgiDown_30 AT %MX30212.30 : BOOL;
	bSlowPull1LifterStn3AgiDown_31 AT %MX30212.31 : BOOL;

	bSlowPull1LifterStn4AgiDown_00 AT %MX30216.0 : BOOL;
	bSlowPull1LifterStn4AgiDown_01 AT %MX30216.1 : BOOL;
	bSlowPull1LifterStn4AgiDown_02 AT %MX30216.2 : BOOL;
	bSlowPull1LifterStn4AgiDown_03 AT %MX30216.3 : BOOL;
	bSlowPull1LifterStn4AgiDown_04 AT %MX30216.4 : BOOL;
	bSlowPull1LifterStn4AgiDown_05 AT %MX30216.5 : BOOL;
	bSlowPull1LifterStn4AgiDown_06 AT %MX30216.6 : BOOL;
	bSlowPull1LifterStn4AgiDown_07 AT %MX30216.7 : BOOL;
	bSlowPull1LifterStn4AgiDown_08 AT %MX30216.8 : BOOL;
	bSlowPull1LifterStn4AgiDown_09 AT %MX30216.9 : BOOL;
	bSlowPull1LifterStn4AgiDown_10 AT %MX30216.10 : BOOL;
	bSlowPull1LifterStn4AgiDown_11 AT %MX30216.11 : BOOL;
	bSlowPull1LifterStn4AgiDown_12 AT %MX30216.12 : BOOL;
	bSlowPull1LifterStn4AgiDown_13 AT %MX30216.13 : BOOL;
	bSlowPull1LifterStn4AgiDown_14 AT %MX30216.14 : BOOL;
	bSlowPull1LifterStn4AgiDown_15 AT %MX30216.15 : BOOL;
	bSlowPull1LifterStn4AgiDown_16 AT %MX30216.16 : BOOL;
	bSlowPull1LifterStn4AgiDown_17 AT %MX30216.17 : BOOL;
	bSlowPull1LifterStn4AgiDown_18 AT %MX30216.18 : BOOL;
	bSlowPull1LifterStn4AgiDown_19 AT %MX30216.19 : BOOL;
	bSlowPull1LifterStn4AgiDown_20 AT %MX30216.20 : BOOL;
	bSlowPull1LifterStn4AgiDown_21 AT %MX30216.21 : BOOL;
	bSlowPull1LifterStn4AgiDown_22 AT %MX30216.22 : BOOL;
	bSlowPull1LifterStn4AgiDown_23 AT %MX30216.23 : BOOL;
	bSlowPull1LifterStn4AgiDown_24 AT %MX30216.24 : BOOL;
	bSlowPull1LifterStn4AgiDown_25 AT %MX30216.25 : BOOL;
	bSlowPull1LifterStn4AgiDown_26 AT %MX30216.26 : BOOL;
	bSlowPull1LifterStn4AgiDown_27 AT %MX30216.27 : BOOL;
	bSlowPull1LifterStn4AgiDown_28 AT %MX30216.28 : BOOL;
	bSlowPull1LifterStn4AgiDown_29 AT %MX30216.29 : BOOL;
	bSlowPull1LifterStn4AgiDown_30 AT %MX30216.30 : BOOL;
	bSlowPull1LifterStn4AgiDown_31 AT %MX30216.31 : BOOL;

	bSlowPull1LifterStn5AgiDown_00 AT %MX30220.0 : BOOL;
	bSlowPull1LifterStn5AgiDown_01 AT %MX30220.1 : BOOL;
	bSlowPull1LifterStn5AgiDown_02 AT %MX30220.2 : BOOL;
	bSlowPull1LifterStn5AgiDown_03 AT %MX30220.3 : BOOL;
	bSlowPull1LifterStn5AgiDown_04 AT %MX30220.4 : BOOL;
	bSlowPull1LifterStn5AgiDown_05 AT %MX30220.5 : BOOL;
	bSlowPull1LifterStn5AgiDown_06 AT %MX30220.6 : BOOL;
	bSlowPull1LifterStn5AgiDown_07 AT %MX30220.7 : BOOL;
	bSlowPull1LifterStn5AgiDown_08 AT %MX30220.8 : BOOL;
	bSlowPull1LifterStn5AgiDown_09 AT %MX30220.9 : BOOL;
	bSlowPull1LifterStn5AgiDown_10 AT %MX30220.10 : BOOL;
	bSlowPull1LifterStn5AgiDown_11 AT %MX30220.11 : BOOL;
	bSlowPull1LifterStn5AgiDown_12 AT %MX30220.12 : BOOL;
	bSlowPull1LifterStn5AgiDown_13 AT %MX30220.13 : BOOL;
	bSlowPull1LifterStn5AgiDown_14 AT %MX30220.14 : BOOL;
	bSlowPull1LifterStn5AgiDown_15 AT %MX30220.15 : BOOL;
	bSlowPull1LifterStn5AgiDown_16 AT %MX30220.16 : BOOL;
	bSlowPull1LifterStn5AgiDown_17 AT %MX30220.17 : BOOL;
	bSlowPull1LifterStn5AgiDown_18 AT %MX30220.18 : BOOL;
	bSlowPull1LifterStn5AgiDown_19 AT %MX30220.19 : BOOL;
	bSlowPull1LifterStn5AgiDown_20 AT %MX30220.20 : BOOL;
	bSlowPull1LifterStn5AgiDown_21 AT %MX30220.21 : BOOL;
	bSlowPull1LifterStn5AgiDown_22 AT %MX30220.22 : BOOL;
	bSlowPull1LifterStn5AgiDown_23 AT %MX30220.23 : BOOL;
	bSlowPull1LifterStn5AgiDown_24 AT %MX30220.24 : BOOL;
	bSlowPull1LifterStn5AgiDown_25 AT %MX30220.25 : BOOL;
	bSlowPull1LifterStn5AgiDown_26 AT %MX30220.26 : BOOL;
	bSlowPull1LifterStn5AgiDown_27 AT %MX30220.27 : BOOL;
	bSlowPull1LifterStn5AgiDown_28 AT %MX30220.28 : BOOL;
	bSlowPull1LifterStn5AgiDown_29 AT %MX30220.29 : BOOL;
	bSlowPull1LifterStn5AgiDown_30 AT %MX30220.30 : BOOL;
	bSlowPull1LifterStn5AgiDown_31 AT %MX30220.31 : BOOL;

	bSlowPull1LifterStn6AgiDown_00 AT %MX30224.0 : BOOL;
	bSlowPull1LifterStn6AgiDown_01 AT %MX30224.1 : BOOL;
	bSlowPull1LifterStn6AgiDown_02 AT %MX30224.2 : BOOL;
	bSlowPull1LifterStn6AgiDown_03 AT %MX30224.3 : BOOL;
	bSlowPull1LifterStn6AgiDown_04 AT %MX30224.4 : BOOL;
	bSlowPull1LifterStn6AgiDown_05 AT %MX30224.5 : BOOL;
	bSlowPull1LifterStn6AgiDown_06 AT %MX30224.6 : BOOL;
	bSlowPull1LifterStn6AgiDown_07 AT %MX30224.7 : BOOL;
	bSlowPull1LifterStn6AgiDown_08 AT %MX30224.8 : BOOL;
	bSlowPull1LifterStn6AgiDown_09 AT %MX30224.9 : BOOL;
	bSlowPull1LifterStn6AgiDown_10 AT %MX30224.10 : BOOL;
	bSlowPull1LifterStn6AgiDown_11 AT %MX30224.11 : BOOL;
	bSlowPull1LifterStn6AgiDown_12 AT %MX30224.12 : BOOL;
	bSlowPull1LifterStn6AgiDown_13 AT %MX30224.13 : BOOL;
	bSlowPull1LifterStn6AgiDown_14 AT %MX30224.14 : BOOL;
	bSlowPull1LifterStn6AgiDown_15 AT %MX30224.15 : BOOL;
	bSlowPull1LifterStn6AgiDown_16 AT %MX30224.16 : BOOL;
	bSlowPull1LifterStn6AgiDown_17 AT %MX30224.17 : BOOL;
	bSlowPull1LifterStn6AgiDown_18 AT %MX30224.18 : BOOL;
	bSlowPull1LifterStn6AgiDown_19 AT %MX30224.19 : BOOL;
	bSlowPull1LifterStn6AgiDown_20 AT %MX30224.20 : BOOL;
	bSlowPull1LifterStn6AgiDown_21 AT %MX30224.21 : BOOL;
	bSlowPull1LifterStn6AgiDown_22 AT %MX30224.22 : BOOL;
	bSlowPull1LifterStn6AgiDown_23 AT %MX30224.23 : BOOL;
	bSlowPull1LifterStn6AgiDown_24 AT %MX30224.24 : BOOL;
	bSlowPull1LifterStn6AgiDown_25 AT %MX30224.25 : BOOL;
	bSlowPull1LifterStn6AgiDown_26 AT %MX30224.26 : BOOL;
	bSlowPull1LifterStn6AgiDown_27 AT %MX30224.27 : BOOL;
	bSlowPull1LifterStn6AgiDown_28 AT %MX30224.28 : BOOL;
	bSlowPull1LifterStn6AgiDown_29 AT %MX30224.29 : BOOL;
	bSlowPull1LifterStn6AgiDown_30 AT %MX30224.30 : BOOL;
	bSlowPull1LifterStn6AgiDown_31 AT %MX30224.31 : BOOL;

	bSlowPull1LifterStn7AgiDown_00 AT %MX30228.0 : BOOL;
	bSlowPull1LifterStn7AgiDown_01 AT %MX30228.1 : BOOL;
	bSlowPull1LifterStn7AgiDown_02 AT %MX30228.2 : BOOL;
	bSlowPull1LifterStn7AgiDown_03 AT %MX30228.3 : BOOL;
	bSlowPull1LifterStn7AgiDown_04 AT %MX30228.4 : BOOL;
	bSlowPull1LifterStn7AgiDown_05 AT %MX30228.5 : BOOL;
	bSlowPull1LifterStn7AgiDown_06 AT %MX30228.6 : BOOL;
	bSlowPull1LifterStn7AgiDown_07 AT %MX30228.7 : BOOL;
	bSlowPull1LifterStn7AgiDown_08 AT %MX30228.8 : BOOL;
	bSlowPull1LifterStn7AgiDown_09 AT %MX30228.9 : BOOL;
	bSlowPull1LifterStn7AgiDown_10 AT %MX30228.10 : BOOL;
	bSlowPull1LifterStn7AgiDown_11 AT %MX30228.11 : BOOL;
	bSlowPull1LifterStn7AgiDown_12 AT %MX30228.12 : BOOL;
	bSlowPull1LifterStn7AgiDown_13 AT %MX30228.13 : BOOL;
	bSlowPull1LifterStn7AgiDown_14 AT %MX30228.14 : BOOL;
	bSlowPull1LifterStn7AgiDown_15 AT %MX30228.15 : BOOL;
	bSlowPull1LifterStn7AgiDown_16 AT %MX30228.16 : BOOL;
	bSlowPull1LifterStn7AgiDown_17 AT %MX30228.17 : BOOL;
	bSlowPull1LifterStn7AgiDown_18 AT %MX30228.18 : BOOL;
	bSlowPull1LifterStn7AgiDown_19 AT %MX30228.19 : BOOL;
	bSlowPull1LifterStn7AgiDown_20 AT %MX30228.20 : BOOL;
	bSlowPull1LifterStn7AgiDown_21 AT %MX30228.21 : BOOL;
	bSlowPull1LifterStn7AgiDown_22 AT %MX30228.22 : BOOL;
	bSlowPull1LifterStn7AgiDown_23 AT %MX30228.23 : BOOL;
	bSlowPull1LifterStn7AgiDown_24 AT %MX30228.24 : BOOL;
	bSlowPull1LifterStn7AgiDown_25 AT %MX30228.25 : BOOL;
	bSlowPull1LifterStn7AgiDown_26 AT %MX30228.26 : BOOL;
	bSlowPull1LifterStn7AgiDown_27 AT %MX30228.27 : BOOL;
	bSlowPull1LifterStn7AgiDown_28 AT %MX30228.28 : BOOL;
	bSlowPull1LifterStn7AgiDown_29 AT %MX30228.29 : BOOL;
	bSlowPull1LifterStn7AgiDown_30 AT %MX30228.30 : BOOL;
	bSlowPull1LifterStn7AgiDown_31 AT %MX30228.31 : BOOL;

	bSlowPull1LifterStn8AgiDown_00 AT %MX30232.0 : BOOL;
	bSlowPull1LifterStn8AgiDown_01 AT %MX30232.1 : BOOL;
	bSlowPull1LifterStn8AgiDown_02 AT %MX30232.2 : BOOL;
	bSlowPull1LifterStn8AgiDown_03 AT %MX30232.3 : BOOL;
	bSlowPull1LifterStn8AgiDown_04 AT %MX30232.4 : BOOL;
	bSlowPull1LifterStn8AgiDown_05 AT %MX30232.5 : BOOL;
	bSlowPull1LifterStn8AgiDown_06 AT %MX30232.6 : BOOL;
	bSlowPull1LifterStn8AgiDown_07 AT %MX30232.7 : BOOL;
	bSlowPull1LifterStn8AgiDown_08 AT %MX30232.8 : BOOL;
	bSlowPull1LifterStn8AgiDown_09 AT %MX30232.9 : BOOL;
	bSlowPull1LifterStn8AgiDown_10 AT %MX30232.10 : BOOL;
	bSlowPull1LifterStn8AgiDown_11 AT %MX30232.11 : BOOL;
	bSlowPull1LifterStn8AgiDown_12 AT %MX30232.12 : BOOL;
	bSlowPull1LifterStn8AgiDown_13 AT %MX30232.13 : BOOL;
	bSlowPull1LifterStn8AgiDown_14 AT %MX30232.14 : BOOL;
	bSlowPull1LifterStn8AgiDown_15 AT %MX30232.15 : BOOL;
	bSlowPull1LifterStn8AgiDown_16 AT %MX30232.16 : BOOL;
	bSlowPull1LifterStn8AgiDown_17 AT %MX30232.17 : BOOL;
	bSlowPull1LifterStn8AgiDown_18 AT %MX30232.18 : BOOL;
	bSlowPull1LifterStn8AgiDown_19 AT %MX30232.19 : BOOL;
	bSlowPull1LifterStn8AgiDown_20 AT %MX30232.20 : BOOL;
	bSlowPull1LifterStn8AgiDown_21 AT %MX30232.21 : BOOL;
	bSlowPull1LifterStn8AgiDown_22 AT %MX30232.22 : BOOL;
	bSlowPull1LifterStn8AgiDown_23 AT %MX30232.23 : BOOL;
	bSlowPull1LifterStn8AgiDown_24 AT %MX30232.24 : BOOL;
	bSlowPull1LifterStn8AgiDown_25 AT %MX30232.25 : BOOL;
	bSlowPull1LifterStn8AgiDown_26 AT %MX30232.26 : BOOL;
	bSlowPull1LifterStn8AgiDown_27 AT %MX30232.27 : BOOL;
	bSlowPull1LifterStn8AgiDown_28 AT %MX30232.28 : BOOL;
	bSlowPull1LifterStn8AgiDown_29 AT %MX30232.29 : BOOL;
	bSlowPull1LifterStn8AgiDown_30 AT %MX30232.30 : BOOL;
	bSlowPull1LifterStn8AgiDown_31 AT %MX30232.31 : BOOL;

	bSlowPull1LifterStn9AgiDown_00 AT %MX30236.0 : BOOL;
	bSlowPull1LifterStn9AgiDown_01 AT %MX30236.1 : BOOL;
	bSlowPull1LifterStn9AgiDown_02 AT %MX30236.2 : BOOL;
	bSlowPull1LifterStn9AgiDown_03 AT %MX30236.3 : BOOL;
	bSlowPull1LifterStn9AgiDown_04 AT %MX30236.4 : BOOL;
	bSlowPull1LifterStn9AgiDown_05 AT %MX30236.5 : BOOL;
	bSlowPull1LifterStn9AgiDown_06 AT %MX30236.6 : BOOL;
	bSlowPull1LifterStn9AgiDown_07 AT %MX30236.7 : BOOL;
	bSlowPull1LifterStn9AgiDown_08 AT %MX30236.8 : BOOL;
	bSlowPull1LifterStn9AgiDown_09 AT %MX30236.9 : BOOL;
	bSlowPull1LifterStn9AgiDown_10 AT %MX30236.10 : BOOL;
	bSlowPull1LifterStn9AgiDown_11 AT %MX30236.11 : BOOL;
	bSlowPull1LifterStn9AgiDown_12 AT %MX30236.12 : BOOL;
	bSlowPull1LifterStn9AgiDown_13 AT %MX30236.13 : BOOL;
	bSlowPull1LifterStn9AgiDown_14 AT %MX30236.14 : BOOL;
	bSlowPull1LifterStn9AgiDown_15 AT %MX30236.15 : BOOL;
	bSlowPull1LifterStn9AgiDown_16 AT %MX30236.16 : BOOL;
	bSlowPull1LifterStn9AgiDown_17 AT %MX30236.17 : BOOL;
	bSlowPull1LifterStn9AgiDown_18 AT %MX30236.18 : BOOL;
	bSlowPull1LifterStn9AgiDown_19 AT %MX30236.19 : BOOL;
	bSlowPull1LifterStn9AgiDown_20 AT %MX30236.20 : BOOL;
	bSlowPull1LifterStn9AgiDown_21 AT %MX30236.21 : BOOL;
	bSlowPull1LifterStn9AgiDown_22 AT %MX30236.22 : BOOL;
	bSlowPull1LifterStn9AgiDown_23 AT %MX30236.23 : BOOL;
	bSlowPull1LifterStn9AgiDown_24 AT %MX30236.24 : BOOL;
	bSlowPull1LifterStn9AgiDown_25 AT %MX30236.25 : BOOL;
	bSlowPull1LifterStn9AgiDown_26 AT %MX30236.26 : BOOL;
	bSlowPull1LifterStn9AgiDown_27 AT %MX30236.27 : BOOL;
	bSlowPull1LifterStn9AgiDown_28 AT %MX30236.28 : BOOL;
	bSlowPull1LifterStn9AgiDown_29 AT %MX30236.29 : BOOL;
	bSlowPull1LifterStn9AgiDown_30 AT %MX30236.30 : BOOL;
	bSlowPull1LifterStn9AgiDown_31 AT %MX30236.31 : BOOL;

